// TIA Portal V19 export
FUNCTION_BLOCK "Generic_FB"   // FB108, LAD
TITLE = GENERIC STUFF OF AREA 01 CONTROL CABINET
// stored: Access Published, MemoryReserve 100, SetENOAutomatically false
   VAR_INPUT
      AreaInterface1 : "AreaInterface";
      AreaInterface2 : "AreaInterface";
      AreaInterface3 : "AreaInterface";
      AreaInterface4 : "AreaInterface";
   END_VAR
   VAR_OUTPUT
      MachineInterface1 : "MachineInterface";
      MachineInterface2 : "MachineInterface";
      MachineInterface3 : "MachineInterface";
      MachineInterface4 : "MachineInterface";
   END_VAR
   VAR
      Ctrl : Struct
         RstAlarms : Bool;
      END_STRUCT;
      Sts : Struct
         Standstill : Bool := TRUE;
         AlarmsPresence_GEN : Bool := FALSE;
         AlarmsPresence_A01_2 : Bool;
         AlarmsPresence_A03_4 : Bool;
         WarningsPresence : Bool := FALSE;
      END_STRUCT;
      Alarm : Struct
         CC1_PorteAperte : Bool;
         CC1_ThermalTrip_24Vdc_PLC_SINAMICS : Bool;
         CC1_ThermalTrip_24Vdc_Valves : Bool;
         CC1_ProtezioneElettronicaSitop : Bool;
         CC1_LowAirPressure : Bool;
         Area01_Aspo_LowAirPressure : Bool;
         Area02_03_Accopiamento_LowAirPressure : Bool;
         Area03_Pareggiamneto_LowAirPressure : Bool;
         Area04_Navetta_LowAirPressure : Bool;
         INFEED_640A1 : "InfeedAlr";
         CU_580A1 : "SinamicsCU_Alarms";
         CU_585A1 : "SinamicsCU_Alarms";
         CU_590A1 : "SinamicsCU_Alarms";
         CU_595A1 : "SinamicsCU_Alarms";
         CU_600A1 : "SinamicsCU_Alarms";
         CU_605A1 : "SinamicsCU_Alarms";
         CU_610A1 : "SinamicsCU_Alarms";
         CU_615A1 : "SinamicsCU_Alarms";
         PNDiag_ET200S_460A1 : "PnDiag_Alr";
         PNDiag_ET200S_490A1 : "PnDiag_Alr";
         PNDiag_ET200S_510A1 : "PnDiag_Alr";
         PNDiag_ET200S_530A1 : "PnDiag_Alr";
         PNDiag_ET200S_550A1 : "PnDiag_Alr";
         PNDiag_CU_580A1 : "PnDiag_Alr";
         PNDiag_CU_585A1 : "PnDiag_Alr";
         PNDiag_CU_590A1 : "PnDiag_Alr";
         PNDiag_CU_595A1 : "PnDiag_Alr";
         PNDiag_CU_600A1 : "PnDiag_Alr";
         PNDiag_CU_605A1 : "PnDiag_Alr";
         PNDiag_CU_610A1 : "PnDiag_Alr";
         PNDiag_CU_615A1 : "PnDiag_Alr";
         PnDiag_ENC_694P1 { S7_SetPoint := 'True'} : "PnDiag_Alr";
         PnDiag_ENC_894P1 { S7_SetPoint := 'True'} : "PnDiag_Alr";
         PnDiag_ENC_984P1 { S7_SetPoint := 'True'} : "PnDiag_Alr";
         PnDiag_ENC_994P1 { S7_SetPoint := 'True'} : "PnDiag_Alr";
         PnDiag_ENC_1004P1 { S7_SetPoint := 'True'} : "PnDiag_Alr";
         PnDiag_ENC_1008P1 { S7_SetPoint := 'True'} : "PnDiag_Alr";
         PnDiag_ENC_1034P1 { S7_SetPoint := 'True'} : "PnDiag_Alr";
         PnDiag_ENC_1044P1 { S7_SetPoint := 'True'} : "PnDiag_Alr";
         PnDiag_ENC_1074P1 { S7_SetPoint := 'True'} : "PnDiag_Alr";
         PnDiag_ENC_1088P1 { S7_SetPoint := 'True'} : "PnDiag_Alr";
         PnDiag_ENC_1093P1 { S7_SetPoint := 'True'} : "PnDiag_Alr";
         PnDiag_ENC_1124P1 { S7_SetPoint := 'True'} : "PnDiag_Alr";
         PnDiag_ENC_1138P1 { S7_SetPoint := 'True'} : "PnDiag_Alr";
         PnDiag_ENC_1143P1 { S7_SetPoint := 'True'} : "PnDiag_Alr";
         PnDiag_ENC_1844P1 { S7_SetPoint := 'True'} : "PnDiag_Alr";
         PnDiag_ENC_1853P1 { S7_SetPoint := 'True'} : "PnDiag_Alr";
         PnDiag_ENC_1858P1 { S7_SetPoint := 'True'} : "PnDiag_Alr";
         PnDiag_ENC_1863P1 { S7_SetPoint := 'True'} : "PnDiag_Alr";
         PnDiag_ENC_1868P1 { S7_SetPoint := 'True'} : "PnDiag_Alr";
         PnDiag_ENC_1903P1 { S7_SetPoint := 'True'} : "PnDiag_Alr";
         PnDiag_ENC_1908P1 { S7_SetPoint := 'True'} : "PnDiag_Alr";
         PnDiag_ENC_1913P1 { S7_SetPoint := 'True'} : "PnDiag_Alr";
         PnDiag_ENC_1918P1 { S7_SetPoint := 'True'} : "PnDiag_Alr";
         PnDiag_ENC_2264P1 { S7_SetPoint := 'True'} : "PnDiag_Alr";
         PnDiag_ENC_2284P1 { S7_SetPoint := 'True'} : "PnDiag_Alr";
         PnDiag_ENC_2374P1 { S7_SetPoint := 'True'} : "PnDiag_Alr";
         PnDiag_ENC_2394P1 { S7_SetPoint := 'True'} : "PnDiag_Alr";
         PnDiag_ENC_2404P1 { S7_SetPoint := 'True'} : "PnDiag_Alr";
         PnDiag_ENC_2434P1 { S7_SetPoint := 'True'} : "PnDiag_Alr";
         PnDiag_ENC_2464P1 { S7_SetPoint := 'True'} : "PnDiag_Alr";
         PnDiag_ENC_2534P1 { S7_SetPoint := 'True'} : "PnDiag_Alr";
         PnDiag_PAC_100A1 { S7_SetPoint := 'True'} : "PnDiag_Alr";
      END_STRUCT;
      Warning : Struct
         NoAutReady : Bool;
         CC1_ThermalTrip220V_ServiceSockets : Bool;
         CC1_ThermalTrip_Cooling1 : Bool;
         CC1_ThermalTrip_Cooling2 : Bool;
         JB001_ThermalTrip_Cooling : Bool;
         CC1_MaxTemperature : Bool;
         JB001_MaxTemperature : Bool;
         CC1_GuastoCondizionatore_1 : Bool;
         CC1_GuastoCondizionatore_2 : Bool;
         SitopUp_BatteriaScarica : Bool;
         SitopUp_BatteriaNonCarica : Bool;
         SitopUp_AllarmeBatteria : Bool;
         ScalanceXC116_1_NotOk : Bool;
         ScalanceXC116_2_NotOk : Bool;
         ScalanceXC216_NotOk : Bool;
         ScalanceSC632_NotOk : Bool;
         INFEED_640A1 : "InfeedWng";
         CU_580A1 : "SinamicsCU_Warnings";
         CU_585A1 : "SinamicsCU_Warnings";
         CU_590A1 : "SinamicsCU_Warnings";
         CU_595A1 : "SinamicsCU_Warnings";
         CU_600A1 : "SinamicsCU_Warnings";
         CU_605A1 : "SinamicsCU_Warnings";
         CU_610A1 : "SinamicsCU_Warnings";
         CU_615A1 : "SinamicsCU_Warnings";
      END_STRUCT;
      Diag : Struct
         CC1_INFEED_460A1 : "TO_Diagnostic";
         CU_580A1 { S7_SetPoint := 'True'} : "TO_Diagnostic";
         CU_585A1 { S7_SetPoint := 'True'} : "TO_Diagnostic";
         CU_590A1 { S7_SetPoint := 'True'} : "TO_Diagnostic";
         CU_595A1 { S7_SetPoint := 'True'} : "TO_Diagnostic";
         CU_600A1 { S7_SetPoint := 'True'} : "TO_Diagnostic";
         CU_605A1 { S7_SetPoint := 'True'} : "TO_Diagnostic";
         CU_610A1 { S7_SetPoint := 'True'} : "TO_Diagnostic";
         CU_615A1 { S7_SetPoint := 'True'} : "TO_Diagnostic";
      END_STRUCT;
      INFEED_640A1 : "Infeed";
      CU_580A1 : "SinamicsCU_Modulblock";
      CU_585A1 : "SinamicsCU_Modulblock";
      CU_590A1 : "SinamicsCU_Modulblock";
      CU_595A1 : "SinamicsCU_Modulblock";
      CU_600A1 : "SinamicsCU_Modulblock";
      CU_605A1 : "SinamicsCU_Modulblock";
      CU_610A1 : "SinamicsCU_Modulblock";
      CU_615A1 : "SinamicsCU_Modulblock";
      PnDiag_ET200S_460A1 : "PnDiag";
      PnDiag_ET200S_490A1 : "PnDiag";
      PnDiag_ET200S_510A1 : "PnDiag";
      PnDiag_ET200S_530A1 : "PnDiag";
      PnDiag_ET200S_550A1 : "PnDiag";
      PnDiag_CU_580A1 : "PnDiag";
      PnDiag_CU_585A1 : "PnDiag";
      PnDiag_CU_590A1 : "PnDiag";
      PnDiag_CU_595A1 : "PnDiag";
      PnDiag_CU_600A1 : "PnDiag";
      PnDiag_CU_605A1 : "PnDiag";
      PnDiag_CU_610A1 : "PnDiag";
      PnDiag_CU_615A1 : "PnDiag";
      PnDiag_ENC_694P1 { S7_SetPoint := 'True'} : "PnDiag";
      PnDiag_ENC_894P1 { S7_SetPoint := 'True'} : "PnDiag";
      PnDiag_ENC_984P1 { S7_SetPoint := 'True'} : "PnDiag";
      PnDiag_ENC_994P1 { S7_SetPoint := 'True'} : "PnDiag";
      PnDiag_ENC_1004P1 { S7_SetPoint := 'True'} : "PnDiag";
      PnDiag_ENC_1008P1 { S7_SetPoint := 'True'} : "PnDiag";
      PnDiag_ENC_1034P1 { S7_SetPoint := 'True'} : "PnDiag";
      PnDiag_ENC_1044P1 { S7_SetPoint := 'True'} : "PnDiag";
      PnDiag_ENC_1074P1 { S7_SetPoint := 'True'} : "PnDiag";
      PnDiag_ENC_1088P1 { S7_SetPoint := 'True'} : "PnDiag";
      PnDiag_ENC_1093P1 { S7_SetPoint := 'True'} : "PnDiag";
      PnDiag_ENC_1124P1 { S7_SetPoint := 'True'} : "PnDiag";
      PnDiag_ENC_1138P1 { S7_SetPoint := 'True'} : "PnDiag";
      PnDiag_ENC_1143P1 { S7_SetPoint := 'True'} : "PnDiag";
      PnDiag_ENC_1844P1 { S7_SetPoint := 'True'} : "PnDiag";
      PnDiag_ENC_1853P1 { S7_SetPoint := 'True'} : "PnDiag";
      PnDiag_ENC_1858P1 { S7_SetPoint := 'True'} : "PnDiag";
      PnDiag_ENC_1863P1 { S7_SetPoint := 'True'} : "PnDiag";
      PnDiag_ENC_1868P1 { S7_SetPoint := 'True'} : "PnDiag";
      PnDiag_ENC_1903P1 { S7_SetPoint := 'True'} : "PnDiag";
      PnDiag_ENC_1908P1 { S7_SetPoint := 'True'} : "PnDiag";
      PnDiag_ENC_1913P1 { S7_SetPoint := 'True'} : "PnDiag";
      PnDiag_ENC_1918P1 { S7_SetPoint := 'True'} : "PnDiag";
      PnDiag_ENC_2264P1 { S7_SetPoint := 'True'} : "PnDiag";
      PnDiag_ENC_2284P1 { S7_SetPoint := 'True'} : "PnDiag";
      PnDiag_ENC_2374P1 { S7_SetPoint := 'True'} : "PnDiag";
      PnDiag_ENC_2394P1 { S7_SetPoint := 'True'} : "PnDiag";
      PnDiag_ENC_2404P1 { S7_SetPoint := 'True'} : "PnDiag";
      PnDiag_ENC_2434P1 { S7_SetPoint := 'True'} : "PnDiag";
      PnDiag_ENC_2464P1 { S7_SetPoint := 'True'} : "PnDiag";
      PnDiag_ENC_2534P1 { S7_SetPoint := 'True'} : "PnDiag";
      PnDiag_PAC_100A1 { S7_SetPoint := 'True'} : "PnDiag";
      TON_CheckHighTemperatureCC1 : IEC_TIMER;
      TON_CheckHighTemperatureJB001 : IEC_TIMER;
      TOF_TurnOffConditionerCC1 : IEC_TIMER;
      TOF_TurnOffConditionerJB001 : IEC_TIMER;
      TON_Area02_03_Accoppiamento_Pressione_Aria_OK { S7_SetPoint := 'True'} : IEC_TIMER;
      TON_Area03_Pareggiamneto_Pressione_Aria_OK { S7_SetPoint := 'True'} : IEC_TIMER;
      TON_Area04_Navetta_Pressione_Aria_OK { S7_SetPoint := 'True'} : IEC_TIMER;
   END_VAR
   VAR CONSTANT
      MSG_A1073_POWER_ON_REQ_BACKUP_COPY : UInt := 1073;
      MSG_A13030_TRIAL_LICENSE_ACTIVATE : UInt := 13030;
   END_VAR
BEGIN

REGION Network 1: Reset alarms
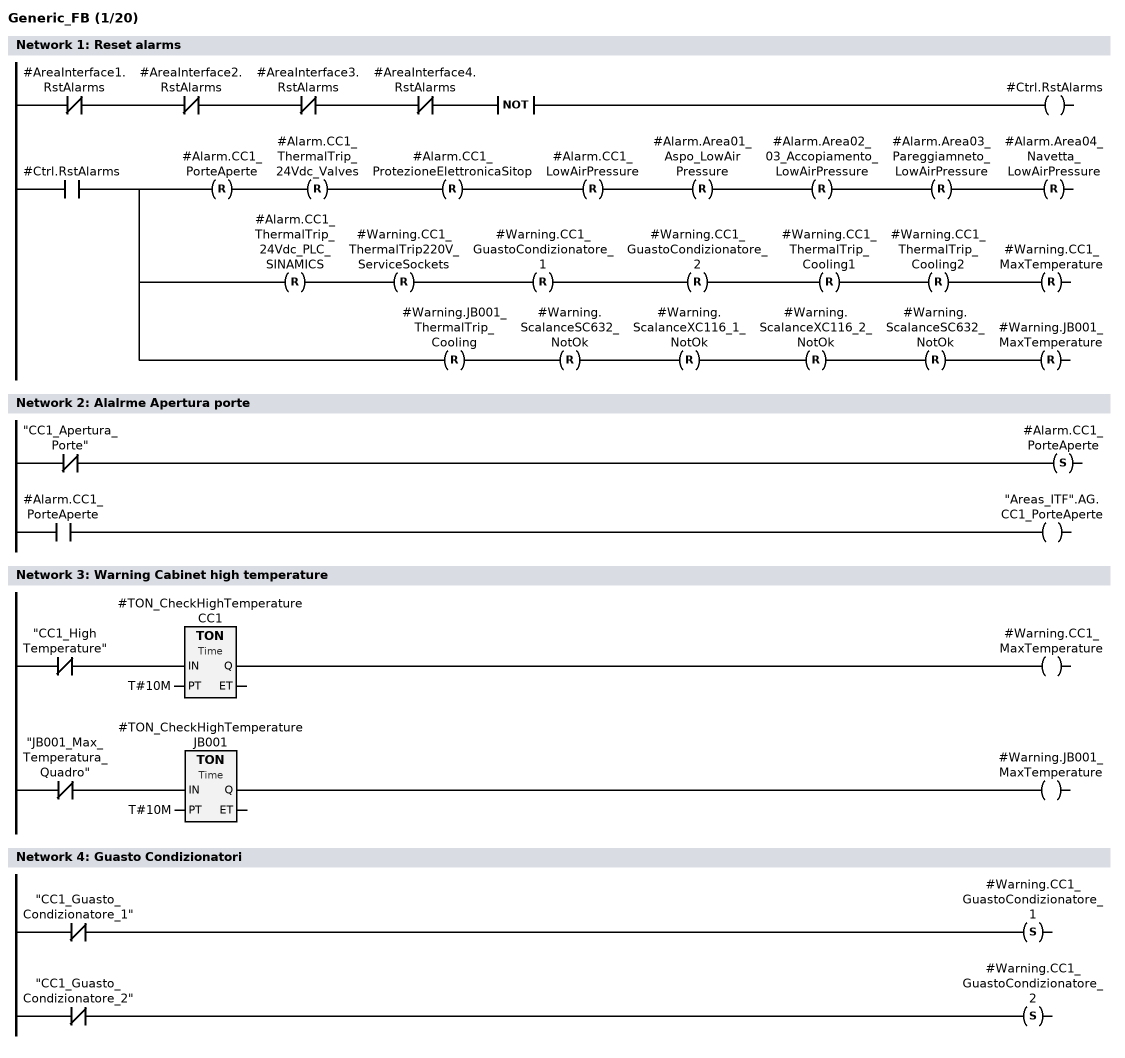
   RUNG wire#powerrail
      I_Contact( #AreaInterface1.RstAlarms )
      I_Contact( #AreaInterface2.RstAlarms )
      I_Contact( #AreaInterface3.RstAlarms )
      I_Contact( #AreaInterface4.RstAlarms )
      Not()
      Coil( #Ctrl.RstAlarms )
   END_RUNG
   RUNG wire#powerrail
      Contact( #Ctrl.RstAlarms )
      wire#w1
      R_Coil( #Alarm.CC1_PorteAperte )
      R_Coil( #Alarm.CC1_ThermalTrip_24Vdc_Valves )
      R_Coil( #Alarm.CC1_ProtezioneElettronicaSitop )
      R_Coil( #Alarm.CC1_LowAirPressure )
      R_Coil( #Alarm.Area01_Aspo_LowAirPressure )
      R_Coil( #Alarm.Area02_03_Accopiamento_LowAirPressure )
      R_Coil( #Alarm.Area03_Pareggiamneto_LowAirPressure )
      R_Coil( #Alarm.Area04_Navetta_LowAirPressure )
   END_RUNG
   RUNG wire#w1
      R_Coil( #Alarm.CC1_ThermalTrip_24Vdc_PLC_SINAMICS )
      R_Coil( #Warning.CC1_ThermalTrip220V_ServiceSockets )
      R_Coil( #Warning.CC1_GuastoCondizionatore_1 )
      R_Coil( #Warning.CC1_GuastoCondizionatore_2 )
      R_Coil( #Warning.CC1_ThermalTrip_Cooling1 )
      R_Coil( #Warning.CC1_ThermalTrip_Cooling2 )
      R_Coil( #Warning.CC1_MaxTemperature )
   END_RUNG
   RUNG wire#w1
      R_Coil( #Warning.JB001_ThermalTrip_Cooling )
      R_Coil( #Warning.ScalanceSC632_NotOk )
      R_Coil( #Warning.ScalanceXC116_1_NotOk )
      R_Coil( #Warning.ScalanceXC116_2_NotOk )
      R_Coil( #Warning.ScalanceSC632_NotOk )
      R_Coil( #Warning.JB001_MaxTemperature )
   END_RUNG
   // the same network as SCL:
   #Ctrl.RstAlarms := NOT (NOT #AreaInterface1.RstAlarms AND NOT #AreaInterface2.RstAlarms AND NOT #AreaInterface3.RstAlarms AND NOT #AreaInterface4.RstAlarms);
   IF #Ctrl.RstAlarms THEN
       #Alarm.CC1_PorteAperte := FALSE;
       #Alarm.CC1_ThermalTrip_24Vdc_Valves := FALSE;
       #Alarm.CC1_ProtezioneElettronicaSitop := FALSE;
       #Alarm.CC1_LowAirPressure := FALSE;
       #Alarm.Area01_Aspo_LowAirPressure := FALSE;
       #Alarm.Area02_03_Accopiamento_LowAirPressure := FALSE;
       #Alarm.Area03_Pareggiamneto_LowAirPressure := FALSE;
       #Alarm.Area04_Navetta_LowAirPressure := FALSE;
       #Alarm.CC1_ThermalTrip_24Vdc_PLC_SINAMICS := FALSE;
       #Warning.CC1_ThermalTrip220V_ServiceSockets := FALSE;
       #Warning.CC1_GuastoCondizionatore_1 := FALSE;
       #Warning.CC1_GuastoCondizionatore_2 := FALSE;
       #Warning.CC1_ThermalTrip_Cooling1 := FALSE;
       #Warning.CC1_ThermalTrip_Cooling2 := FALSE;
       #Warning.CC1_MaxTemperature := FALSE;
       #Warning.JB001_ThermalTrip_Cooling := FALSE;
       #Warning.ScalanceSC632_NotOk := FALSE;
       #Warning.ScalanceXC116_1_NotOk := FALSE;
       #Warning.ScalanceXC116_2_NotOk := FALSE;
       #Warning.ScalanceSC632_NotOk := FALSE;
       #Warning.JB001_MaxTemperature := FALSE;
   END_IF;
END_REGION

REGION Network 2: Alalrme Apertura porte
   RUNG wire#powerrail
      I_Contact( "CC1_Apertura_Porte" )
      S_Coil( #Alarm.CC1_PorteAperte )
   END_RUNG
   RUNG wire#powerrail
      Contact( #Alarm.CC1_PorteAperte )
      Coil( "Areas_ITF".AG.CC1_PorteAperte )
   END_RUNG
   // the same network as SCL:
   IF NOT "CC1_Apertura_Porte" THEN #Alarm.CC1_PorteAperte := TRUE; END_IF;
   "Areas_ITF".AG.CC1_PorteAperte := #Alarm.CC1_PorteAperte;
END_REGION

REGION Network 3: Warning Cabinet high temperature
   RUNG wire#powerrail
      I_Contact( "CC1_HighTemperature" )
      { S7_Templates := "time_type := Time" } #TON_CheckHighTemperatureCC1.TON(pt := T#10M, et =>)
      Coil( #Warning.CC1_MaxTemperature )
   END_RUNG
   RUNG wire#powerrail
      I_Contact( "JB001_Max_Temperatura_Quadro" )
      { S7_Templates := "time_type := Time" } #TON_CheckHighTemperatureJB001.TON(pt := T#10M, et =>)
      Coil( #Warning.JB001_MaxTemperature )
   END_RUNG
   // the same network as SCL:
   #TON_CheckHighTemperatureCC1.TON(IN := NOT "CC1_HighTemperature", PT := T#10M);
   #Warning.CC1_MaxTemperature := #TON_CheckHighTemperatureCC1.Q;
   #TON_CheckHighTemperatureJB001.TON(IN := NOT "JB001_Max_Temperatura_Quadro", PT := T#10M);
   #Warning.JB001_MaxTemperature := #TON_CheckHighTemperatureJB001.Q;
END_REGION

REGION Network 4: Guasto Condizionatori
   RUNG wire#powerrail
      I_Contact( "CC1_Guasto_Condizionatore_1" )
      S_Coil( #Warning.CC1_GuastoCondizionatore_1 )
   END_RUNG
   RUNG wire#powerrail
      I_Contact( "CC1_Guasto_Condizionatore_2" )
      S_Coil( #Warning.CC1_GuastoCondizionatore_2 )
   END_RUNG
   // the same network as SCL:
   IF NOT "CC1_Guasto_Condizionatore_1" THEN #Warning.CC1_GuastoCondizionatore_1 := TRUE; END_IF;
   IF NOT "CC1_Guasto_Condizionatore_2" THEN #Warning.CC1_GuastoCondizionatore_2 := TRUE; END_IF;
END_REGION

REGION Network 5: Comando Condizionatori
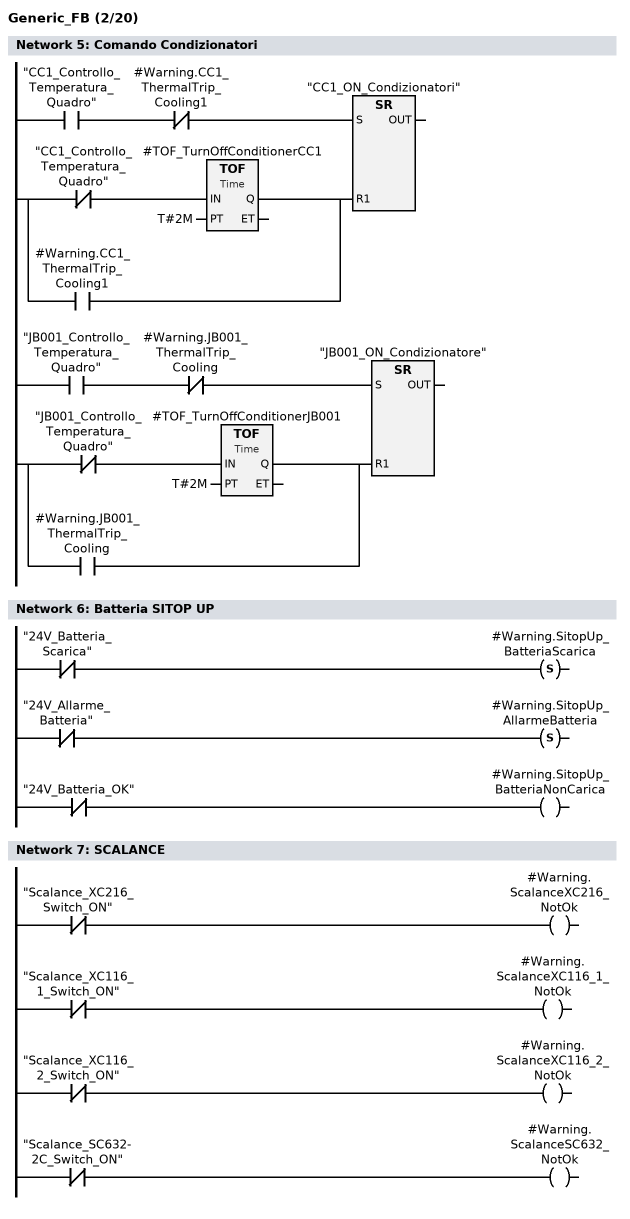
   RUNG wire#powerrail
      Contact( "CC1_Controllo_Temperatura_Quadro" )
      I_Contact( #Warning.CC1_ThermalTrip_Cooling1 )
      S_SR(operand := "CC1_ON_Condizionatori", r1 := wire#w1)
   END_RUNG
   RUNG wire#powerrail
      I_Contact( "CC1_Controllo_Temperatura_Quadro" )
      { S7_Templates := "time_type := Time" } #TOF_TurnOffConditionerCC1.TOF(pt := T#2M, et =>)
   END_RUNG wire#w1
   RUNG wire#powerrail
      Contact( #Warning.CC1_ThermalTrip_Cooling1 )
   END_RUNG wire#w1
   RUNG wire#powerrail
      Contact( "JB001_Controllo_Temperatura_Quadro" )
      I_Contact( #Warning.JB001_ThermalTrip_Cooling )
      S_SR(operand := "JB001_ON_Condizionatore", r1 := wire#w2)
   END_RUNG
   RUNG wire#powerrail
      I_Contact( "JB001_Controllo_Temperatura_Quadro" )
      { S7_Templates := "time_type := Time" } #TOF_TurnOffConditionerJB001.TOF(pt := T#2M, et =>)
   END_RUNG wire#w2
   RUNG wire#powerrail
      Contact( #Warning.JB001_ThermalTrip_Cooling )
   END_RUNG wire#w2
   // the same network as SCL:
   #TOF_TurnOffConditionerCC1.TOF(IN := NOT "CC1_Controllo_Temperatura_Quadro", PT := T#2M);
   IF "CC1_Controllo_Temperatura_Quadro" AND NOT #Warning.CC1_ThermalTrip_Cooling1 THEN
       "CC1_ON_Condizionatori" := TRUE;   // SR flip-flop
   END_IF;
   IF #TOF_TurnOffConditionerCC1.Q OR #Warning.CC1_ThermalTrip_Cooling1 THEN
       "CC1_ON_Condizionatori" := FALSE;
   END_IF;
   #TOF_TurnOffConditionerJB001.TOF(IN := NOT "JB001_Controllo_Temperatura_Quadro", PT := T#2M);
   IF "JB001_Controllo_Temperatura_Quadro" AND NOT #Warning.JB001_ThermalTrip_Cooling THEN
       "JB001_ON_Condizionatore" := TRUE;   // SR flip-flop
   END_IF;
   IF #TOF_TurnOffConditionerJB001.Q OR #Warning.JB001_ThermalTrip_Cooling THEN
       "JB001_ON_Condizionatore" := FALSE;
   END_IF;
END_REGION

REGION Network 6: Batteria SITOP UP
   RUNG wire#powerrail
      I_Contact( "24V_Batteria_Scarica" )
      S_Coil( #Warning.SitopUp_BatteriaScarica )
   END_RUNG
   RUNG wire#powerrail
      I_Contact( "24V_Allarme_Batteria" )
      S_Coil( #Warning.SitopUp_AllarmeBatteria )
   END_RUNG
   RUNG wire#powerrail
      I_Contact( "24V_Batteria_OK" )
      Coil( #Warning.SitopUp_BatteriaNonCarica )
   END_RUNG
   // the same network as SCL:
   IF NOT "24V_Batteria_Scarica" THEN #Warning.SitopUp_BatteriaScarica := TRUE; END_IF;
   IF NOT "24V_Allarme_Batteria" THEN #Warning.SitopUp_AllarmeBatteria := TRUE; END_IF;
   #Warning.SitopUp_BatteriaNonCarica := NOT "24V_Batteria_OK";
END_REGION

REGION Network 7: SCALANCE
   RUNG wire#powerrail
      I_Contact( "Scalance_XC216_Switch_ON" )
      Coil( #Warning.ScalanceXC216_NotOk )
   END_RUNG
   RUNG wire#powerrail
      I_Contact( "Scalance_XC116_1_Switch_ON" )
      Coil( #Warning.ScalanceXC116_1_NotOk )
   END_RUNG
   RUNG wire#powerrail
      I_Contact( "Scalance_XC116_2_Switch_ON" )
      Coil( #Warning.ScalanceXC116_2_NotOk )
   END_RUNG
   RUNG wire#powerrail
      I_Contact( "Scalance_SC632-2C_Switch_ON" )
      Coil( #Warning.ScalanceSC632_NotOk )
   END_RUNG
   // the same network as SCL:
   #Warning.ScalanceXC216_NotOk := NOT "Scalance_XC216_Switch_ON";
   #Warning.ScalanceXC116_1_NotOk := NOT "Scalance_XC116_1_Switch_ON";
   #Warning.ScalanceXC116_2_NotOk := NOT "Scalance_XC116_2_Switch_ON";
   #Warning.ScalanceSC632_NotOk := NOT "Scalance_SC632-2C_Switch_ON";
END_REGION

REGION Network 8: Alarm Thermal trips
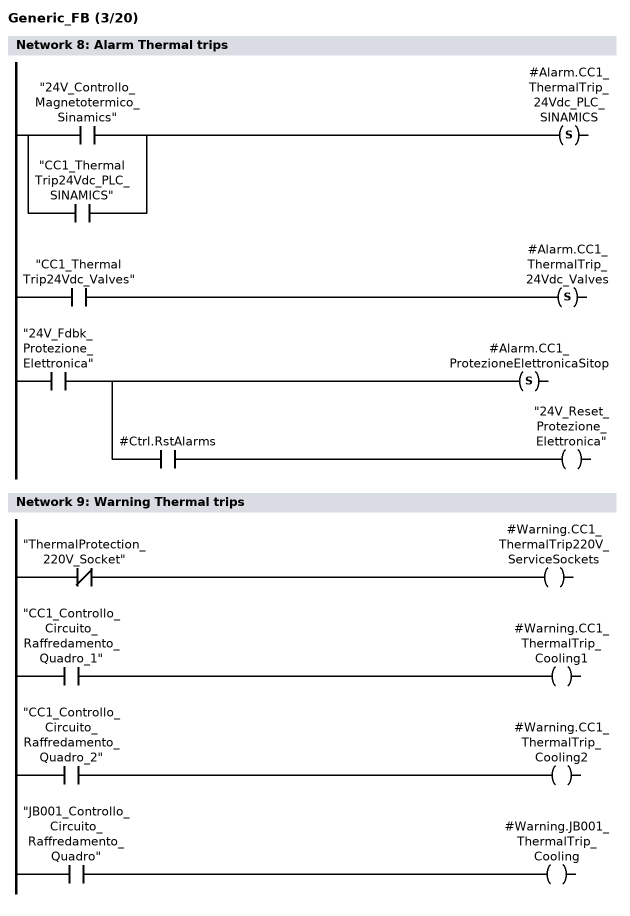
   RUNG wire#powerrail
      Contact( "24V_Controllo_Magnetotermico_Sinamics" )
      wire#w1
      S_Coil( #Alarm.CC1_ThermalTrip_24Vdc_PLC_SINAMICS )
   END_RUNG
   RUNG wire#powerrail
      Contact( "CC1_ThermalTrip24Vdc_PLC_SINAMICS" )
   END_RUNG wire#w1
   RUNG wire#powerrail
      Contact( "CC1_ThermalTrip24Vdc_Valves" )
      S_Coil( #Alarm.CC1_ThermalTrip_24Vdc_Valves )
   END_RUNG
   RUNG wire#powerrail
      Contact( "24V_Fdbk_Protezione_Elettronica" )
      wire#w2
      S_Coil( #Alarm.CC1_ProtezioneElettronicaSitop )
   END_RUNG
   RUNG wire#w2
      Contact( #Ctrl.RstAlarms )
      Coil( "24V_Reset_Protezione_Elettronica" )
   END_RUNG
   // the same network as SCL:
   IF "24V_Controllo_Magnetotermico_Sinamics" OR "CC1_ThermalTrip24Vdc_PLC_SINAMICS" THEN
       #Alarm.CC1_ThermalTrip_24Vdc_PLC_SINAMICS := TRUE;
   END_IF;
   IF "CC1_ThermalTrip24Vdc_Valves" THEN #Alarm.CC1_ThermalTrip_24Vdc_Valves := TRUE; END_IF;
   IF "24V_Fdbk_Protezione_Elettronica" THEN #Alarm.CC1_ProtezioneElettronicaSitop := TRUE; END_IF;
   "24V_Reset_Protezione_Elettronica" := "24V_Fdbk_Protezione_Elettronica" AND #Ctrl.RstAlarms;
END_REGION

REGION Network 9: Warning Thermal trips
   RUNG wire#powerrail
      I_Contact( "ThermalProtection_220V_Socket" )
      Coil( #Warning.CC1_ThermalTrip220V_ServiceSockets )
   END_RUNG
   RUNG wire#powerrail
      Contact( "CC1_Controllo_Circuito_Raffredamento_Quadro_1" )
      Coil( #Warning.CC1_ThermalTrip_Cooling1 )
   END_RUNG
   RUNG wire#powerrail
      Contact( "CC1_Controllo_Circuito_Raffredamento_Quadro_2" )
      Coil( #Warning.CC1_ThermalTrip_Cooling2 )
   END_RUNG
   RUNG wire#powerrail
      Contact( "JB001_Controllo_Circuito_Raffredamento_Quadro" )
      Coil( #Warning.JB001_ThermalTrip_Cooling )
   END_RUNG
   // the same network as SCL:
   #Warning.CC1_ThermalTrip220V_ServiceSockets := NOT "ThermalProtection_220V_Socket";
   #Warning.CC1_ThermalTrip_Cooling1 := "CC1_Controllo_Circuito_Raffredamento_Quadro_1";
   #Warning.CC1_ThermalTrip_Cooling2 := "CC1_Controllo_Circuito_Raffredamento_Quadro_2";
   #Warning.JB001_ThermalTrip_Cooling := "JB001_Controllo_Circuito_Raffredamento_Quadro";
END_REGION

REGION Network 10: Alarm Low air pressure
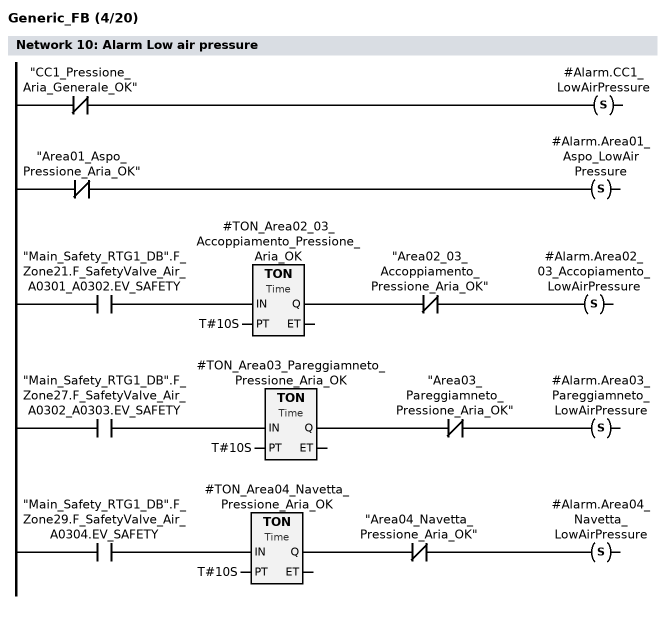
   RUNG wire#powerrail
      I_Contact( "CC1_Pressione_Aria_Generale_OK" )
      S_Coil( #Alarm.CC1_LowAirPressure )
   END_RUNG
   RUNG wire#powerrail
      I_Contact( "Area01_Aspo_Pressione_Aria_OK" )
      S_Coil( #Alarm.Area01_Aspo_LowAirPressure )
   END_RUNG
   RUNG wire#powerrail
      Contact( "Main_Safety_RTG1_DB".F_Zone21.F_SafetyValve_Air_A0301_A0302.EV_SAFETY )
      { S7_Templates := "time_type := Time" } #TON_Area02_03_Accoppiamento_Pressione_Aria_OK.TON(pt := T#10S, et =>)
      I_Contact( "Area02_03_Accoppiamento_Pressione_Aria_OK" )
      S_Coil( #Alarm.Area02_03_Accopiamento_LowAirPressure )
   END_RUNG
   RUNG wire#powerrail
      Contact( "Main_Safety_RTG1_DB".F_Zone27.F_SafetyValve_Air_A0302_A0303.EV_SAFETY )
      { S7_Templates := "time_type := Time" } #TON_Area03_Pareggiamneto_Pressione_Aria_OK.TON(pt := T#10S, et =>)
      I_Contact( "Area03_Pareggiamneto_Pressione_Aria_OK" )
      S_Coil( #Alarm.Area03_Pareggiamneto_LowAirPressure )
   END_RUNG
   RUNG wire#powerrail
      Contact( "Main_Safety_RTG1_DB".F_Zone29.F_SafetyValve_Air_A0304.EV_SAFETY )
      { S7_Templates := "time_type := Time" } #TON_Area04_Navetta_Pressione_Aria_OK.TON(pt := T#10S, et =>)
      I_Contact( "Area04_Navetta_Pressione_Aria_OK" )
      S_Coil( #Alarm.Area04_Navetta_LowAirPressure )
   END_RUNG
   // the same network as SCL:
   IF NOT "CC1_Pressione_Aria_Generale_OK" THEN #Alarm.CC1_LowAirPressure := TRUE; END_IF;
   IF NOT "Area01_Aspo_Pressione_Aria_OK" THEN #Alarm.Area01_Aspo_LowAirPressure := TRUE; END_IF;
   #TON_Area02_03_Accoppiamento_Pressione_Aria_OK.TON(IN := "Main_Safety_RTG1_DB".F_Zone21.F_SafetyValve_Air_A0301_A0302.EV_SAFETY,
                           PT := T#10S);
   IF #TON_Area02_03_Accoppiamento_Pressione_Aria_OK.Q AND NOT "Area02_03_Accoppiamento_Pressione_Aria_OK" THEN
       #Alarm.Area02_03_Accopiamento_LowAirPressure := TRUE;
   END_IF;
   #TON_Area03_Pareggiamneto_Pressione_Aria_OK.TON(IN := "Main_Safety_RTG1_DB".F_Zone27.F_SafetyValve_Air_A0302_A0303.EV_SAFETY,
                           PT := T#10S);
   IF #TON_Area03_Pareggiamneto_Pressione_Aria_OK.Q AND NOT "Area03_Pareggiamneto_Pressione_Aria_OK" THEN
       #Alarm.Area03_Pareggiamneto_LowAirPressure := TRUE;
   END_IF;
   #TON_Area04_Navetta_Pressione_Aria_OK.TON(IN := "Main_Safety_RTG1_DB".F_Zone29.F_SafetyValve_Air_A0304.EV_SAFETY,
                           PT := T#10S);
   IF #TON_Area04_Navetta_Pressione_Aria_OK.Q AND NOT "Area04_Navetta_Pressione_Aria_OK" THEN
       #Alarm.Area04_Navetta_LowAirPressure := TRUE;
   END_IF;
END_REGION

REGION Network 12: <<< DRIVES >>>
END_REGION

REGION Network 13: Infeed
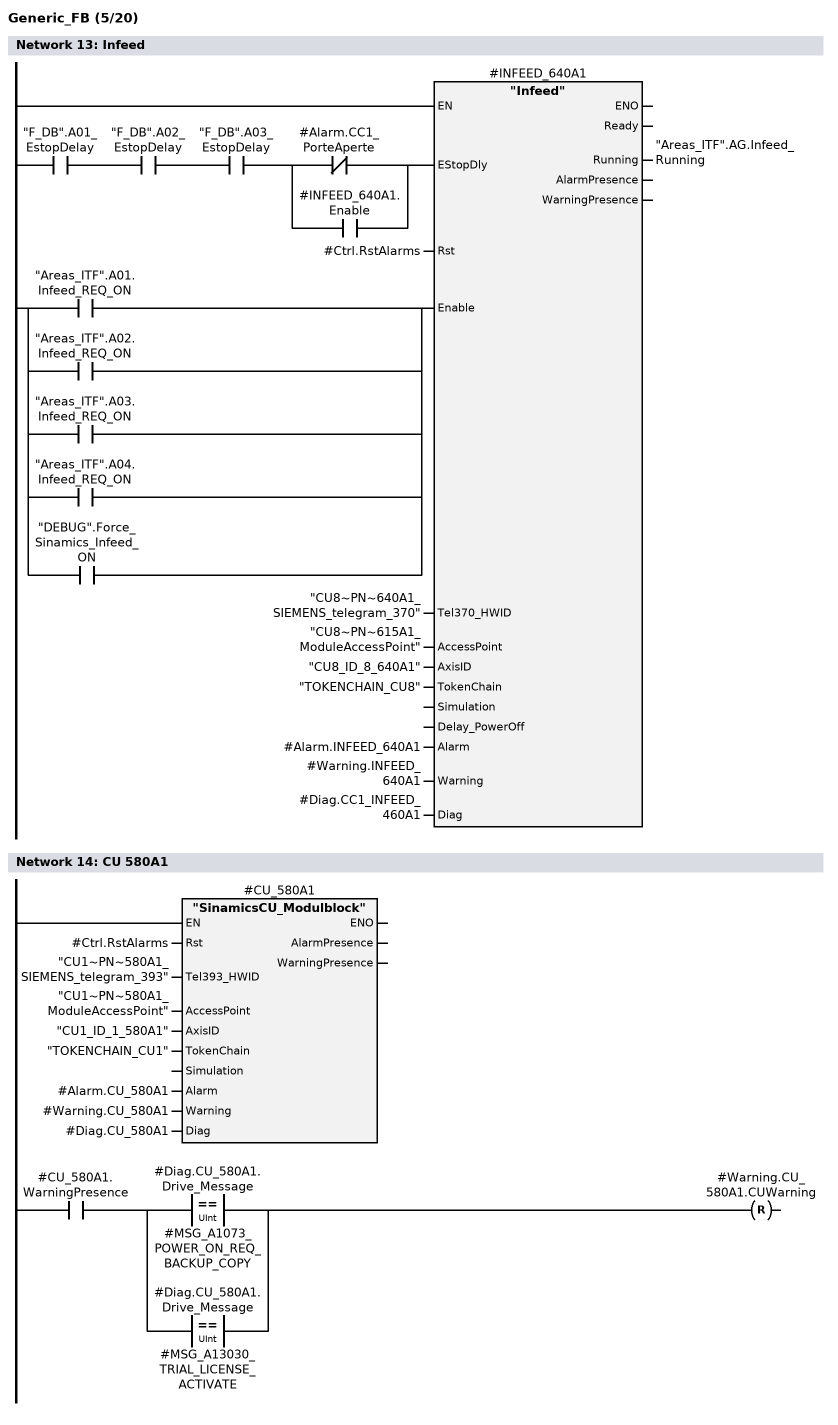
   RUNG wire#powerrail
      #INFEED_640A1(EStopDly := wire#w2, Enable := wire#w3, Rst := #Ctrl.RstAlarms, Tel370_HWID := "CU8~PN~640A1_SIEMENS_telegram_370", AccessPoint := "CU8~PN~615A1_ModuleAccessPoint", AxisID := "CU8_ID_8_640A1", TokenChain := "TOKENCHAIN_CU8", Simulation :=, Delay_PowerOff :=, Alarm := #Alarm.INFEED_640A1, Warning := #Warning.INFEED_640A1, Diag := #Diag.CC1_INFEED_460A1, Ready =>, Running => "Areas_ITF".AG.Infeed_Running, AlarmPresence =>, WarningPresence =>)
   END_RUNG
   RUNG wire#powerrail
      Contact( "F_DB".A01_EstopDelay )
      Contact( "F_DB".A02_EstopDelay )
      Contact( "F_DB".A03_EstopDelay )
      wire#w1
      I_Contact( #Alarm.CC1_PorteAperte )
   END_RUNG wire#w2
   RUNG wire#w1
      Contact( #INFEED_640A1.Enable )
   END_RUNG wire#w2
   RUNG wire#powerrail
      Contact( "Areas_ITF".A01.Infeed_REQ_ON )
   END_RUNG wire#w3
   RUNG wire#powerrail
      Contact( "Areas_ITF".A02.Infeed_REQ_ON )
   END_RUNG wire#w3
   RUNG wire#powerrail
      Contact( "Areas_ITF".A03.Infeed_REQ_ON )
   END_RUNG wire#w3
   RUNG wire#powerrail
      Contact( "Areas_ITF".A04.Infeed_REQ_ON )
   END_RUNG wire#w3
   RUNG wire#powerrail
      Contact( "DEBUG".Force_Sinamics_Infeed_ON )
   END_RUNG wire#w3
   // the same network as SCL:
   #INFEED_640A1(EStopDly := "F_DB".A01_EstopDelay AND "F_DB".A02_EstopDelay AND "F_DB".A03_EstopDelay AND (NOT #Alarm.CC1_PorteAperte OR #INFEED_640A1.Enable),   // "Infeed"
                 Rst := #Ctrl.RstAlarms,
                 Enable := "Areas_ITF".A01.Infeed_REQ_ON OR "Areas_ITF".A02.Infeed_REQ_ON OR "Areas_ITF".A03.Infeed_REQ_ON OR "Areas_ITF".A04.Infeed_REQ_ON OR "DEBUG".Force_Sinamics_Infeed_ON,
                 Tel370_HWID := "CU8~PN~640A1_SIEMENS_telegram_370",
                 AccessPoint := "CU8~PN~615A1_ModuleAccessPoint",
                 AxisID := "CU8_ID_8_640A1",
                 TokenChain := "TOKENCHAIN_CU8",
                 Alarm := #Alarm.INFEED_640A1,
                 Warning := #Warning.INFEED_640A1,
                 Diag := #Diag.CC1_INFEED_460A1,
                 Running => "Areas_ITF".AG.Infeed_Running);
END_REGION

REGION Network 14: CU 580A1
   RUNG wire#powerrail
      #CU_580A1(Rst := #Ctrl.RstAlarms, Tel393_HWID := "CU1~PN~580A1_SIEMENS_telegram_393", AccessPoint := "CU1~PN~580A1_ModuleAccessPoint", AxisID := "CU1_ID_1_580A1", TokenChain := "TOKENCHAIN_CU1", Simulation :=, Alarm := #Alarm.CU_580A1, Warning := #Warning.CU_580A1, Diag := #Diag.CU_580A1, AlarmPresence =>, WarningPresence =>)
   END_RUNG
   RUNG wire#powerrail
      Contact( #CU_580A1.WarningPresence )
      wire#w1
      { S7_Templates := "SrcType := UInt" } EQ_Contact(in1 := #Diag.CU_580A1.Drive_Message, in2 := #MSG_A1073_POWER_ON_REQ_BACKUP_COPY)
      wire#w2
      R_Coil( #Warning.CU_580A1.CUWarning )
   END_RUNG
   RUNG wire#w1
      { S7_Templates := "SrcType := UInt" } EQ_Contact(in1 := #Diag.CU_580A1.Drive_Message, in2 := #MSG_A13030_TRIAL_LICENSE_ACTIVATE)
   END_RUNG wire#w2
   // the same network as SCL:
   #CU_580A1(Rst := #Ctrl.RstAlarms,   // "SinamicsCU_Modulblock"
             Tel393_HWID := "CU1~PN~580A1_SIEMENS_telegram_393",
             AccessPoint := "CU1~PN~580A1_ModuleAccessPoint",
             AxisID := "CU1_ID_1_580A1",
             TokenChain := "TOKENCHAIN_CU1",
             Alarm := #Alarm.CU_580A1,
             Warning := #Warning.CU_580A1,
             Diag := #Diag.CU_580A1);
   IF #CU_580A1.WarningPresence AND ((#Diag.CU_580A1.Drive_Message = #MSG_A1073_POWER_ON_REQ_BACKUP_COPY) OR (#Diag.CU_580A1.Drive_Message = #MSG_A13030_TRIAL_LICENSE_ACTIVATE)) THEN
       #Warning.CU_580A1.CUWarning := FALSE;
   END_IF;
END_REGION

REGION Network 15: CU 585A1
   // Bypass message "POWER ON REQUIRED FOR COPY ON MEMORY CARD"
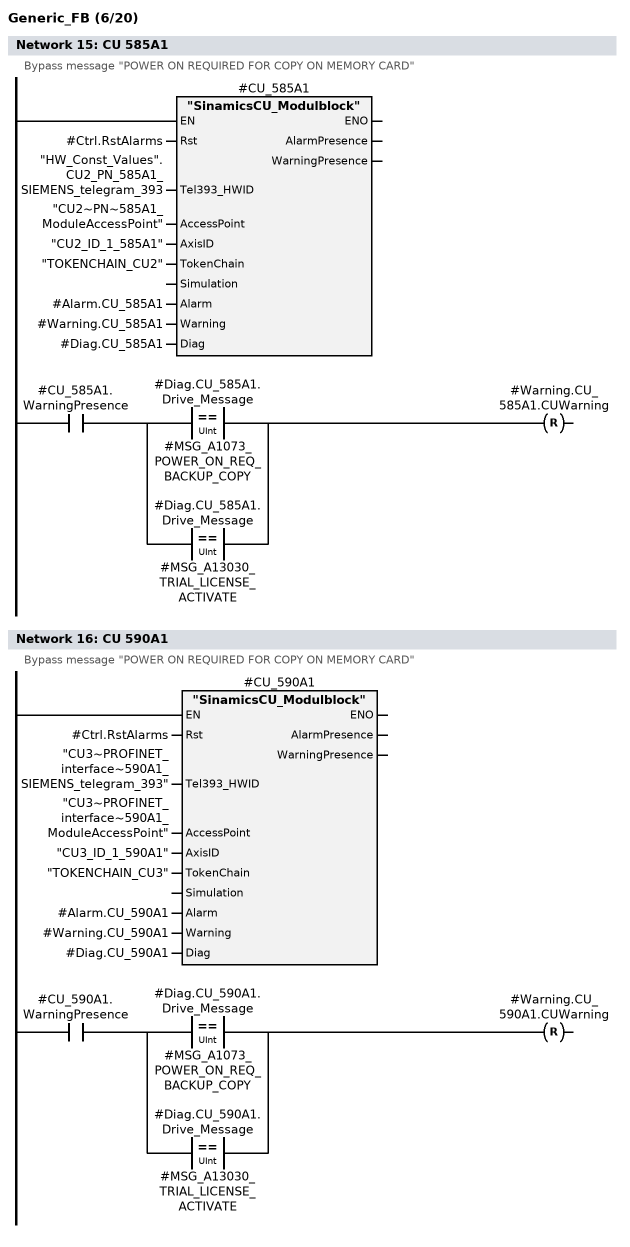
   RUNG wire#powerrail
      #CU_585A1(Rst := #Ctrl.RstAlarms, Tel393_HWID := "HW_Const_Values".CU2_PN_585A1_SIEMENS_telegram_393, AccessPoint := "CU2~PN~585A1_ModuleAccessPoint", AxisID := "CU2_ID_1_585A1", TokenChain := "TOKENCHAIN_CU2", Simulation :=, Alarm := #Alarm.CU_585A1, Warning := #Warning.CU_585A1, Diag := #Diag.CU_585A1, AlarmPresence =>, WarningPresence =>)
   END_RUNG
   RUNG wire#powerrail
      Contact( #CU_585A1.WarningPresence )
      wire#w1
      { S7_Templates := "SrcType := UInt" } EQ_Contact(in1 := #Diag.CU_585A1.Drive_Message, in2 := #MSG_A1073_POWER_ON_REQ_BACKUP_COPY)
      wire#w2
      R_Coil( #Warning.CU_585A1.CUWarning )
   END_RUNG
   RUNG wire#w1
      { S7_Templates := "SrcType := UInt" } EQ_Contact(in1 := #Diag.CU_585A1.Drive_Message, in2 := #MSG_A13030_TRIAL_LICENSE_ACTIVATE)
   END_RUNG wire#w2
   // the same network as SCL:
   #CU_585A1(Rst := #Ctrl.RstAlarms,   // "SinamicsCU_Modulblock"
             Tel393_HWID := "HW_Const_Values".CU2_PN_585A1_SIEMENS_telegram_393,
             AccessPoint := "CU2~PN~585A1_ModuleAccessPoint",
             AxisID := "CU2_ID_1_585A1",
             TokenChain := "TOKENCHAIN_CU2",
             Alarm := #Alarm.CU_585A1,
             Warning := #Warning.CU_585A1,
             Diag := #Diag.CU_585A1);
   IF #CU_585A1.WarningPresence AND ((#Diag.CU_585A1.Drive_Message = #MSG_A1073_POWER_ON_REQ_BACKUP_COPY) OR (#Diag.CU_585A1.Drive_Message = #MSG_A13030_TRIAL_LICENSE_ACTIVATE)) THEN
       #Warning.CU_585A1.CUWarning := FALSE;
   END_IF;
END_REGION

REGION Network 16: CU 590A1
   // Bypass message "POWER ON REQUIRED FOR COPY ON MEMORY CARD"
   RUNG wire#powerrail
      #CU_590A1(Rst := #Ctrl.RstAlarms, Tel393_HWID := "CU3~PROFINET_interface~590A1_SIEMENS_telegram_393", AccessPoint := "CU3~PROFINET_interface~590A1_ModuleAccessPoint", AxisID := "CU3_ID_1_590A1", TokenChain := "TOKENCHAIN_CU3", Simulation :=, Alarm := #Alarm.CU_590A1, Warning := #Warning.CU_590A1, Diag := #Diag.CU_590A1, AlarmPresence =>, WarningPresence =>)
   END_RUNG
   RUNG wire#powerrail
      Contact( #CU_590A1.WarningPresence )
      wire#w1
      { S7_Templates := "SrcType := UInt" } EQ_Contact(in1 := #Diag.CU_590A1.Drive_Message, in2 := #MSG_A1073_POWER_ON_REQ_BACKUP_COPY)
      wire#w2
      R_Coil( #Warning.CU_590A1.CUWarning )
   END_RUNG
   RUNG wire#w1
      { S7_Templates := "SrcType := UInt" } EQ_Contact(in1 := #Diag.CU_590A1.Drive_Message, in2 := #MSG_A13030_TRIAL_LICENSE_ACTIVATE)
   END_RUNG wire#w2
   // the same network as SCL:
   #CU_590A1(Rst := #Ctrl.RstAlarms,   // "SinamicsCU_Modulblock"
             Tel393_HWID := "CU3~PROFINET_interface~590A1_SIEMENS_telegram_393",
             AccessPoint := "CU3~PROFINET_interface~590A1_ModuleAccessPoint",
             AxisID := "CU3_ID_1_590A1",
             TokenChain := "TOKENCHAIN_CU3",
             Alarm := #Alarm.CU_590A1,
             Warning := #Warning.CU_590A1,
             Diag := #Diag.CU_590A1);
   IF #CU_590A1.WarningPresence AND ((#Diag.CU_590A1.Drive_Message = #MSG_A1073_POWER_ON_REQ_BACKUP_COPY) OR (#Diag.CU_590A1.Drive_Message = #MSG_A13030_TRIAL_LICENSE_ACTIVATE)) THEN
       #Warning.CU_590A1.CUWarning := FALSE;
   END_IF;
END_REGION

REGION Network 17: CU 595A1
   // Bypass message "POWER ON REQUIRED FOR COPY ON MEMORY CARD"
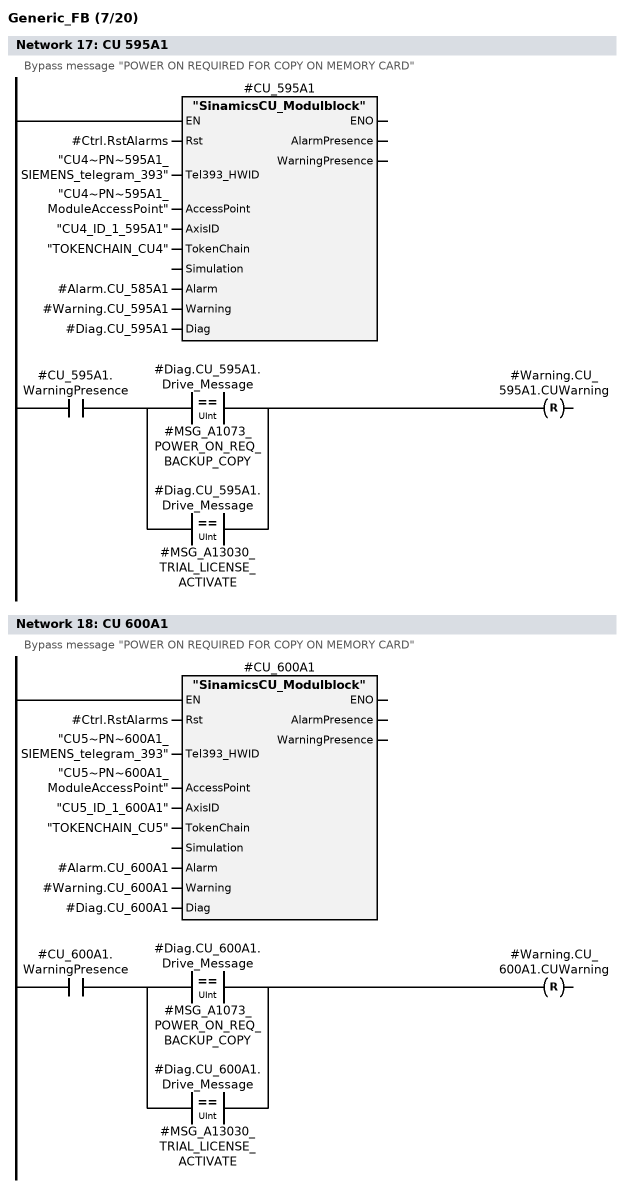
   RUNG wire#powerrail
      #CU_595A1(Rst := #Ctrl.RstAlarms, Tel393_HWID := "CU4~PN~595A1_SIEMENS_telegram_393", AccessPoint := "CU4~PN~595A1_ModuleAccessPoint", AxisID := "CU4_ID_1_595A1", TokenChain := "TOKENCHAIN_CU4", Simulation :=, Alarm := #Alarm.CU_585A1, Warning := #Warning.CU_595A1, Diag := #Diag.CU_595A1, AlarmPresence =>, WarningPresence =>)
   END_RUNG
   RUNG wire#powerrail
      Contact( #CU_595A1.WarningPresence )
      wire#w1
      { S7_Templates := "SrcType := UInt" } EQ_Contact(in1 := #Diag.CU_595A1.Drive_Message, in2 := #MSG_A1073_POWER_ON_REQ_BACKUP_COPY)
      wire#w2
      R_Coil( #Warning.CU_595A1.CUWarning )
   END_RUNG
   RUNG wire#w1
      { S7_Templates := "SrcType := UInt" } EQ_Contact(in1 := #Diag.CU_595A1.Drive_Message, in2 := #MSG_A13030_TRIAL_LICENSE_ACTIVATE)
   END_RUNG wire#w2
   // the same network as SCL:
   #CU_595A1(Rst := #Ctrl.RstAlarms,   // "SinamicsCU_Modulblock"
             Tel393_HWID := "CU4~PN~595A1_SIEMENS_telegram_393",
             AccessPoint := "CU4~PN~595A1_ModuleAccessPoint",
             AxisID := "CU4_ID_1_595A1",
             TokenChain := "TOKENCHAIN_CU4",
             Alarm := #Alarm.CU_585A1,
             Warning := #Warning.CU_595A1,
             Diag := #Diag.CU_595A1);
   IF #CU_595A1.WarningPresence AND ((#Diag.CU_595A1.Drive_Message = #MSG_A1073_POWER_ON_REQ_BACKUP_COPY) OR (#Diag.CU_595A1.Drive_Message = #MSG_A13030_TRIAL_LICENSE_ACTIVATE)) THEN
       #Warning.CU_595A1.CUWarning := FALSE;
   END_IF;
END_REGION

REGION Network 18: CU 600A1
   // Bypass message "POWER ON REQUIRED FOR COPY ON MEMORY CARD"
   RUNG wire#powerrail
      #CU_600A1(Rst := #Ctrl.RstAlarms, Tel393_HWID := "CU5~PN~600A1_SIEMENS_telegram_393", AccessPoint := "CU5~PN~600A1_ModuleAccessPoint", AxisID := "CU5_ID_1_600A1", TokenChain := "TOKENCHAIN_CU5", Simulation :=, Alarm := #Alarm.CU_600A1, Warning := #Warning.CU_600A1, Diag := #Diag.CU_600A1, AlarmPresence =>, WarningPresence =>)
   END_RUNG
   RUNG wire#powerrail
      Contact( #CU_600A1.WarningPresence )
      wire#w1
      { S7_Templates := "SrcType := UInt" } EQ_Contact(in1 := #Diag.CU_600A1.Drive_Message, in2 := #MSG_A1073_POWER_ON_REQ_BACKUP_COPY)
      wire#w2
      R_Coil( #Warning.CU_600A1.CUWarning )
   END_RUNG
   RUNG wire#w1
      { S7_Templates := "SrcType := UInt" } EQ_Contact(in1 := #Diag.CU_600A1.Drive_Message, in2 := #MSG_A13030_TRIAL_LICENSE_ACTIVATE)
   END_RUNG wire#w2
   // the same network as SCL:
   #CU_600A1(Rst := #Ctrl.RstAlarms,   // "SinamicsCU_Modulblock"
             Tel393_HWID := "CU5~PN~600A1_SIEMENS_telegram_393",
             AccessPoint := "CU5~PN~600A1_ModuleAccessPoint",
             AxisID := "CU5_ID_1_600A1",
             TokenChain := "TOKENCHAIN_CU5",
             Alarm := #Alarm.CU_600A1,
             Warning := #Warning.CU_600A1,
             Diag := #Diag.CU_600A1);
   IF #CU_600A1.WarningPresence AND ((#Diag.CU_600A1.Drive_Message = #MSG_A1073_POWER_ON_REQ_BACKUP_COPY) OR (#Diag.CU_600A1.Drive_Message = #MSG_A13030_TRIAL_LICENSE_ACTIVATE)) THEN
       #Warning.CU_600A1.CUWarning := FALSE;
   END_IF;
END_REGION

REGION Network 19: CU 605A1
   // Bypass message "POWER ON REQUIRED FOR COPY ON MEMORY CARD"
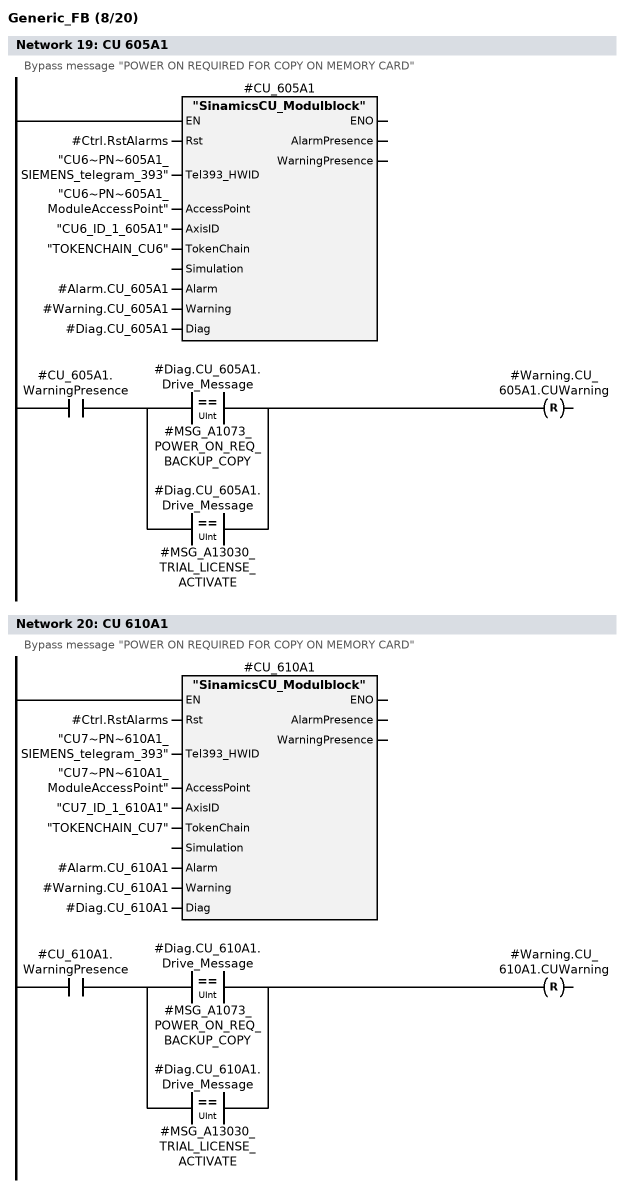
   RUNG wire#powerrail
      #CU_605A1(Rst := #Ctrl.RstAlarms, Tel393_HWID := "CU6~PN~605A1_SIEMENS_telegram_393", AccessPoint := "CU6~PN~605A1_ModuleAccessPoint", AxisID := "CU6_ID_1_605A1", TokenChain := "TOKENCHAIN_CU6", Simulation :=, Alarm := #Alarm.CU_605A1, Warning := #Warning.CU_605A1, Diag := #Diag.CU_605A1, AlarmPresence =>, WarningPresence =>)
   END_RUNG
   RUNG wire#powerrail
      Contact( #CU_605A1.WarningPresence )
      wire#w1
      { S7_Templates := "SrcType := UInt" } EQ_Contact(in1 := #Diag.CU_605A1.Drive_Message, in2 := #MSG_A1073_POWER_ON_REQ_BACKUP_COPY)
      wire#w2
      R_Coil( #Warning.CU_605A1.CUWarning )
   END_RUNG
   RUNG wire#w1
      { S7_Templates := "SrcType := UInt" } EQ_Contact(in1 := #Diag.CU_605A1.Drive_Message, in2 := #MSG_A13030_TRIAL_LICENSE_ACTIVATE)
   END_RUNG wire#w2
   // the same network as SCL:
   #CU_605A1(Rst := #Ctrl.RstAlarms,   // "SinamicsCU_Modulblock"
             Tel393_HWID := "CU6~PN~605A1_SIEMENS_telegram_393",
             AccessPoint := "CU6~PN~605A1_ModuleAccessPoint",
             AxisID := "CU6_ID_1_605A1",
             TokenChain := "TOKENCHAIN_CU6",
             Alarm := #Alarm.CU_605A1,
             Warning := #Warning.CU_605A1,
             Diag := #Diag.CU_605A1);
   IF #CU_605A1.WarningPresence AND ((#Diag.CU_605A1.Drive_Message = #MSG_A1073_POWER_ON_REQ_BACKUP_COPY) OR (#Diag.CU_605A1.Drive_Message = #MSG_A13030_TRIAL_LICENSE_ACTIVATE)) THEN
       #Warning.CU_605A1.CUWarning := FALSE;
   END_IF;
END_REGION

REGION Network 20: CU 610A1
   // Bypass message "POWER ON REQUIRED FOR COPY ON MEMORY CARD"
   RUNG wire#powerrail
      #CU_610A1(Rst := #Ctrl.RstAlarms, Tel393_HWID := "CU7~PN~610A1_SIEMENS_telegram_393", AccessPoint := "CU7~PN~610A1_ModuleAccessPoint", AxisID := "CU7_ID_1_610A1", TokenChain := "TOKENCHAIN_CU7", Simulation :=, Alarm := #Alarm.CU_610A1, Warning := #Warning.CU_610A1, Diag := #Diag.CU_610A1, AlarmPresence =>, WarningPresence =>)
   END_RUNG
   RUNG wire#powerrail
      Contact( #CU_610A1.WarningPresence )
      wire#w1
      { S7_Templates := "SrcType := UInt" } EQ_Contact(in1 := #Diag.CU_610A1.Drive_Message, in2 := #MSG_A1073_POWER_ON_REQ_BACKUP_COPY)
      wire#w2
      R_Coil( #Warning.CU_610A1.CUWarning )
   END_RUNG
   RUNG wire#w1
      { S7_Templates := "SrcType := UInt" } EQ_Contact(in1 := #Diag.CU_610A1.Drive_Message, in2 := #MSG_A13030_TRIAL_LICENSE_ACTIVATE)
   END_RUNG wire#w2
   // the same network as SCL:
   #CU_610A1(Rst := #Ctrl.RstAlarms,   // "SinamicsCU_Modulblock"
             Tel393_HWID := "CU7~PN~610A1_SIEMENS_telegram_393",
             AccessPoint := "CU7~PN~610A1_ModuleAccessPoint",
             AxisID := "CU7_ID_1_610A1",
             TokenChain := "TOKENCHAIN_CU7",
             Alarm := #Alarm.CU_610A1,
             Warning := #Warning.CU_610A1,
             Diag := #Diag.CU_610A1);
   IF #CU_610A1.WarningPresence AND ((#Diag.CU_610A1.Drive_Message = #MSG_A1073_POWER_ON_REQ_BACKUP_COPY) OR (#Diag.CU_610A1.Drive_Message = #MSG_A13030_TRIAL_LICENSE_ACTIVATE)) THEN
       #Warning.CU_610A1.CUWarning := FALSE;
   END_IF;
END_REGION

REGION Network 21: CU 615A1
   // Bypass message "POWER ON REQUIRED FOR COPY ON MEMORY CARD"
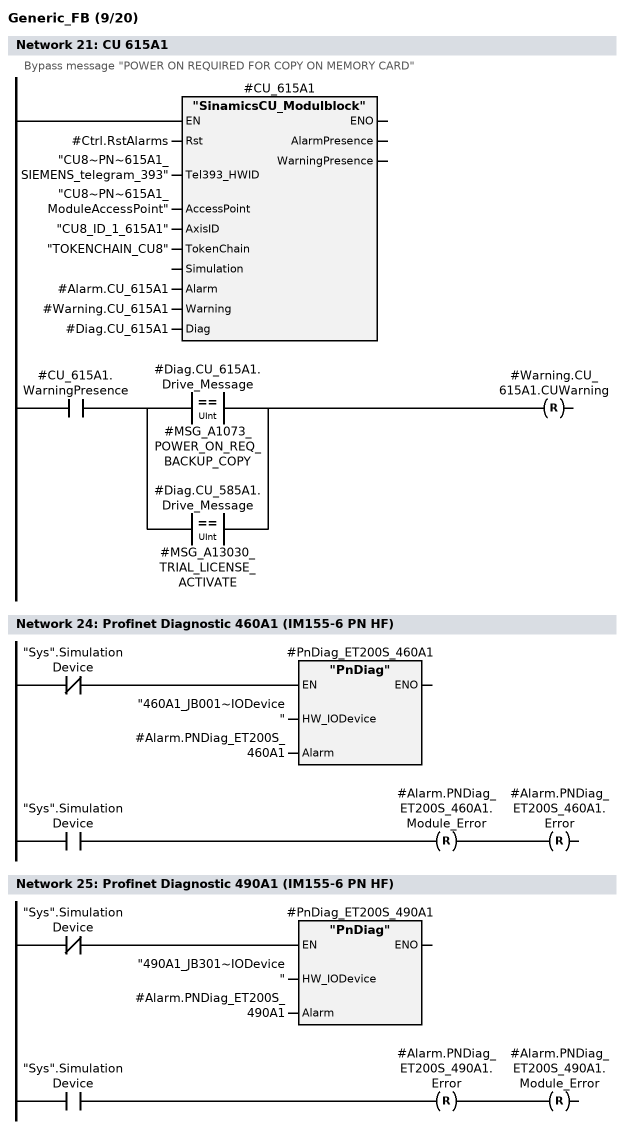
   RUNG wire#powerrail
      #CU_615A1(Rst := #Ctrl.RstAlarms, Tel393_HWID := "CU8~PN~615A1_SIEMENS_telegram_393", AccessPoint := "CU8~PN~615A1_ModuleAccessPoint", AxisID := "CU8_ID_1_615A1", TokenChain := "TOKENCHAIN_CU8", Simulation :=, Alarm := #Alarm.CU_615A1, Warning := #Warning.CU_615A1, Diag := #Diag.CU_615A1, AlarmPresence =>, WarningPresence =>)
   END_RUNG
   RUNG wire#powerrail
      Contact( #CU_615A1.WarningPresence )
      wire#w1
      { S7_Templates := "SrcType := UInt" } EQ_Contact(in1 := #Diag.CU_615A1.Drive_Message, in2 := #MSG_A1073_POWER_ON_REQ_BACKUP_COPY)
      wire#w2
      R_Coil( #Warning.CU_615A1.CUWarning )
   END_RUNG
   RUNG wire#w1
      { S7_Templates := "SrcType := UInt" } EQ_Contact(in1 := #Diag.CU_585A1.Drive_Message, in2 := #MSG_A13030_TRIAL_LICENSE_ACTIVATE)
   END_RUNG wire#w2
   // the same network as SCL:
   #CU_615A1(Rst := #Ctrl.RstAlarms,   // "SinamicsCU_Modulblock"
             Tel393_HWID := "CU8~PN~615A1_SIEMENS_telegram_393",
             AccessPoint := "CU8~PN~615A1_ModuleAccessPoint",
             AxisID := "CU8_ID_1_615A1",
             TokenChain := "TOKENCHAIN_CU8",
             Alarm := #Alarm.CU_615A1,
             Warning := #Warning.CU_615A1,
             Diag := #Diag.CU_615A1);
   IF #CU_615A1.WarningPresence AND ((#Diag.CU_615A1.Drive_Message = #MSG_A1073_POWER_ON_REQ_BACKUP_COPY) OR (#Diag.CU_585A1.Drive_Message = #MSG_A13030_TRIAL_LICENSE_ACTIVATE)) THEN
       #Warning.CU_615A1.CUWarning := FALSE;
   END_IF;
END_REGION

REGION Network 23: <<< PROFINET DIAGNOSTIC >>>
END_REGION

REGION Network 24: Profinet Diagnostic 460A1 (IM155-6 PN HF)
   RUNG wire#powerrail
      I_Contact( "Sys".SimulationDevice )
      #PnDiag_ET200S_460A1(HW_IODevice := "460A1_JB001~IODevice", Alarm := #Alarm.PNDiag_ET200S_460A1)
   END_RUNG
   RUNG wire#powerrail
      Contact( "Sys".SimulationDevice )
      R_Coil( #Alarm.PNDiag_ET200S_460A1.Module_Error )
      R_Coil( #Alarm.PNDiag_ET200S_460A1.Error )
   END_RUNG
   // the same network as SCL:
   IF NOT "Sys".SimulationDevice THEN
       #PnDiag_ET200S_460A1(HW_IODevice := "460A1_JB001~IODevice", Alarm := #Alarm.PNDiag_ET200S_460A1);   // "PnDiag"
   END_IF;
   IF "Sys".SimulationDevice THEN
       #Alarm.PNDiag_ET200S_460A1.Module_Error := FALSE;
       #Alarm.PNDiag_ET200S_460A1.Error := FALSE;
   END_IF;
END_REGION

REGION Network 25: Profinet Diagnostic 490A1 (IM155-6 PN HF)
   RUNG wire#powerrail
      I_Contact( "Sys".SimulationDevice )
      #PnDiag_ET200S_490A1(HW_IODevice := "490A1_JB301~IODevice", Alarm := #Alarm.PNDiag_ET200S_490A1)
   END_RUNG
   RUNG wire#powerrail
      Contact( "Sys".SimulationDevice )
      R_Coil( #Alarm.PNDiag_ET200S_490A1.Error )
      R_Coil( #Alarm.PNDiag_ET200S_490A1.Module_Error )
   END_RUNG
   // the same network as SCL:
   IF NOT "Sys".SimulationDevice THEN
       #PnDiag_ET200S_490A1(HW_IODevice := "490A1_JB301~IODevice", Alarm := #Alarm.PNDiag_ET200S_490A1);   // "PnDiag"
   END_IF;
   IF "Sys".SimulationDevice THEN
       #Alarm.PNDiag_ET200S_490A1.Error := FALSE;
       #Alarm.PNDiag_ET200S_490A1.Module_Error := FALSE;
   END_IF;
END_REGION

REGION Network 26: Profinet Diagnostic 510A1 (IM155-6 PN HF)
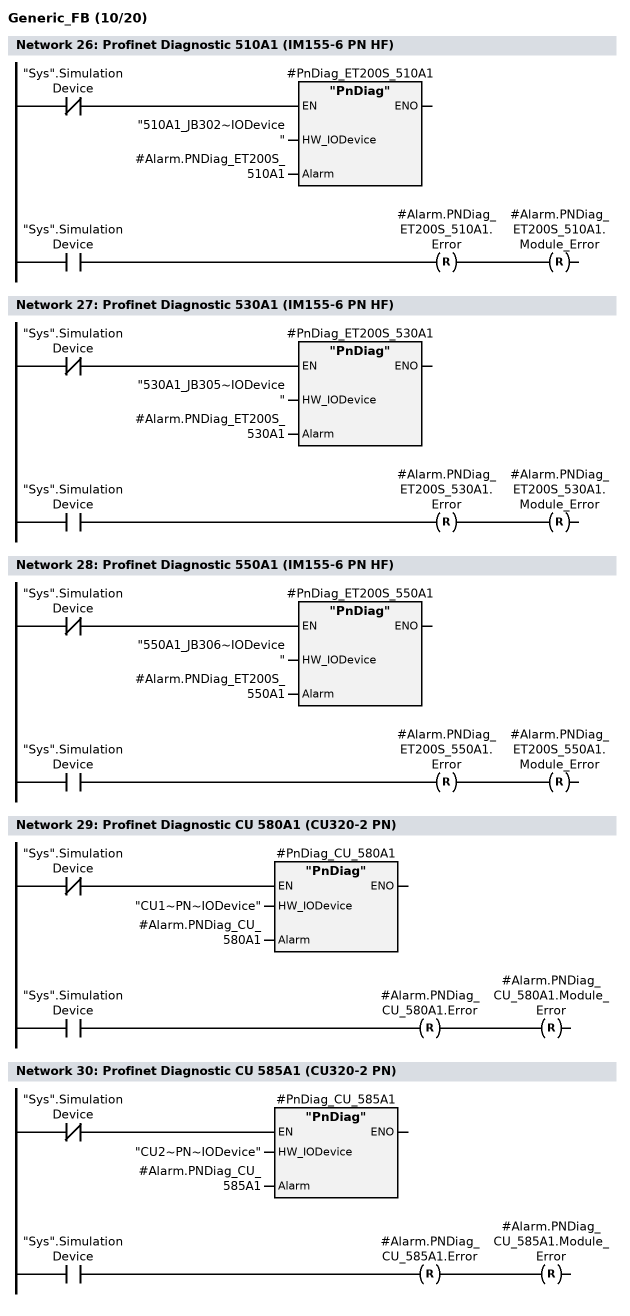
   RUNG wire#powerrail
      I_Contact( "Sys".SimulationDevice )
      #PnDiag_ET200S_510A1(HW_IODevice := "510A1_JB302~IODevice", Alarm := #Alarm.PNDiag_ET200S_510A1)
   END_RUNG
   RUNG wire#powerrail
      Contact( "Sys".SimulationDevice )
      R_Coil( #Alarm.PNDiag_ET200S_510A1.Error )
      R_Coil( #Alarm.PNDiag_ET200S_510A1.Module_Error )
   END_RUNG
   // the same network as SCL:
   IF NOT "Sys".SimulationDevice THEN
       #PnDiag_ET200S_510A1(HW_IODevice := "510A1_JB302~IODevice", Alarm := #Alarm.PNDiag_ET200S_510A1);   // "PnDiag"
   END_IF;
   IF "Sys".SimulationDevice THEN
       #Alarm.PNDiag_ET200S_510A1.Error := FALSE;
       #Alarm.PNDiag_ET200S_510A1.Module_Error := FALSE;
   END_IF;
END_REGION

REGION Network 27: Profinet Diagnostic 530A1 (IM155-6 PN HF)
   RUNG wire#powerrail
      I_Contact( "Sys".SimulationDevice )
      #PnDiag_ET200S_530A1(HW_IODevice := "530A1_JB305~IODevice", Alarm := #Alarm.PNDiag_ET200S_530A1)
   END_RUNG
   RUNG wire#powerrail
      Contact( "Sys".SimulationDevice )
      R_Coil( #Alarm.PNDiag_ET200S_530A1.Error )
      R_Coil( #Alarm.PNDiag_ET200S_530A1.Module_Error )
   END_RUNG
   // the same network as SCL:
   IF NOT "Sys".SimulationDevice THEN
       #PnDiag_ET200S_530A1(HW_IODevice := "530A1_JB305~IODevice", Alarm := #Alarm.PNDiag_ET200S_530A1);   // "PnDiag"
   END_IF;
   IF "Sys".SimulationDevice THEN
       #Alarm.PNDiag_ET200S_530A1.Error := FALSE;
       #Alarm.PNDiag_ET200S_530A1.Module_Error := FALSE;
   END_IF;
END_REGION

REGION Network 28: Profinet Diagnostic 550A1 (IM155-6 PN HF)
   RUNG wire#powerrail
      I_Contact( "Sys".SimulationDevice )
      #PnDiag_ET200S_550A1(HW_IODevice := "550A1_JB306~IODevice", Alarm := #Alarm.PNDiag_ET200S_550A1)
   END_RUNG
   RUNG wire#powerrail
      Contact( "Sys".SimulationDevice )
      R_Coil( #Alarm.PNDiag_ET200S_550A1.Error )
      R_Coil( #Alarm.PNDiag_ET200S_550A1.Module_Error )
   END_RUNG
   // the same network as SCL:
   IF NOT "Sys".SimulationDevice THEN
       #PnDiag_ET200S_550A1(HW_IODevice := "550A1_JB306~IODevice", Alarm := #Alarm.PNDiag_ET200S_550A1);   // "PnDiag"
   END_IF;
   IF "Sys".SimulationDevice THEN
       #Alarm.PNDiag_ET200S_550A1.Error := FALSE;
       #Alarm.PNDiag_ET200S_550A1.Module_Error := FALSE;
   END_IF;
END_REGION

REGION Network 29: Profinet Diagnostic CU 580A1 (CU320-2 PN)
   RUNG wire#powerrail
      I_Contact( "Sys".SimulationDevice )
      #PnDiag_CU_580A1(HW_IODevice := "CU1~PN~IODevice", Alarm := #Alarm.PNDiag_CU_580A1)
   END_RUNG
   RUNG wire#powerrail
      Contact( "Sys".SimulationDevice )
      R_Coil( #Alarm.PNDiag_CU_580A1.Error )
      R_Coil( #Alarm.PNDiag_CU_580A1.Module_Error )
   END_RUNG
   // the same network as SCL:
   IF NOT "Sys".SimulationDevice THEN
       #PnDiag_CU_580A1(HW_IODevice := "CU1~PN~IODevice", Alarm := #Alarm.PNDiag_CU_580A1);   // "PnDiag"
   END_IF;
   IF "Sys".SimulationDevice THEN
       #Alarm.PNDiag_CU_580A1.Error := FALSE;
       #Alarm.PNDiag_CU_580A1.Module_Error := FALSE;
   END_IF;
END_REGION

REGION Network 30: Profinet Diagnostic CU 585A1 (CU320-2 PN)
   RUNG wire#powerrail
      I_Contact( "Sys".SimulationDevice )
      #PnDiag_CU_585A1(HW_IODevice := "CU2~PN~IODevice", Alarm := #Alarm.PNDiag_CU_585A1)
   END_RUNG
   RUNG wire#powerrail
      Contact( "Sys".SimulationDevice )
      R_Coil( #Alarm.PNDiag_CU_585A1.Error )
      R_Coil( #Alarm.PNDiag_CU_585A1.Module_Error )
   END_RUNG
   // the same network as SCL:
   IF NOT "Sys".SimulationDevice THEN
       #PnDiag_CU_585A1(HW_IODevice := "CU2~PN~IODevice", Alarm := #Alarm.PNDiag_CU_585A1);   // "PnDiag"
   END_IF;
   IF "Sys".SimulationDevice THEN
       #Alarm.PNDiag_CU_585A1.Error := FALSE;
       #Alarm.PNDiag_CU_585A1.Module_Error := FALSE;
   END_IF;
END_REGION

REGION Network 31: Profinet Diagnostic CU 590A1 (CU320-2 PN)
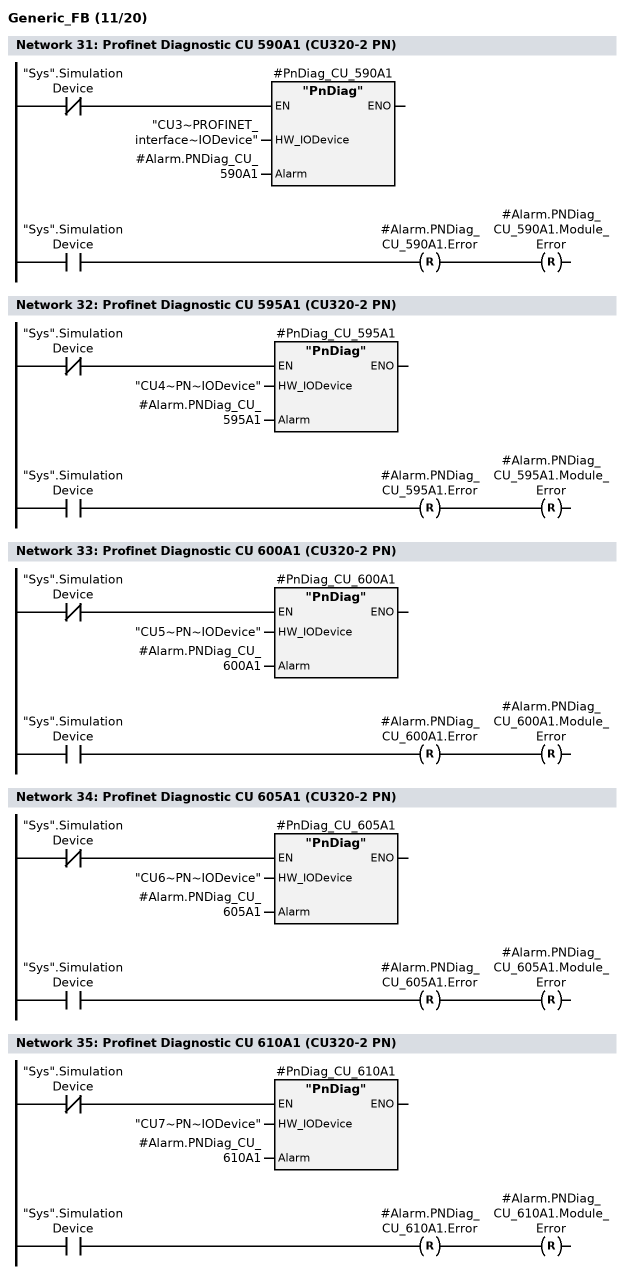
   RUNG wire#powerrail
      I_Contact( "Sys".SimulationDevice )
      #PnDiag_CU_590A1(HW_IODevice := "CU3~PROFINET_interface~IODevice", Alarm := #Alarm.PNDiag_CU_590A1)
   END_RUNG
   RUNG wire#powerrail
      Contact( "Sys".SimulationDevice )
      R_Coil( #Alarm.PNDiag_CU_590A1.Error )
      R_Coil( #Alarm.PNDiag_CU_590A1.Module_Error )
   END_RUNG
   // the same network as SCL:
   IF NOT "Sys".SimulationDevice THEN
       #PnDiag_CU_590A1(HW_IODevice := "CU3~PROFINET_interface~IODevice", Alarm := #Alarm.PNDiag_CU_590A1);   // "PnDiag"
   END_IF;
   IF "Sys".SimulationDevice THEN
       #Alarm.PNDiag_CU_590A1.Error := FALSE;
       #Alarm.PNDiag_CU_590A1.Module_Error := FALSE;
   END_IF;
END_REGION

REGION Network 32: Profinet Diagnostic CU 595A1 (CU320-2 PN)
   RUNG wire#powerrail
      I_Contact( "Sys".SimulationDevice )
      #PnDiag_CU_595A1(HW_IODevice := "CU4~PN~IODevice", Alarm := #Alarm.PNDiag_CU_595A1)
   END_RUNG
   RUNG wire#powerrail
      Contact( "Sys".SimulationDevice )
      R_Coil( #Alarm.PNDiag_CU_595A1.Error )
      R_Coil( #Alarm.PNDiag_CU_595A1.Module_Error )
   END_RUNG
   // the same network as SCL:
   IF NOT "Sys".SimulationDevice THEN
       #PnDiag_CU_595A1(HW_IODevice := "CU4~PN~IODevice", Alarm := #Alarm.PNDiag_CU_595A1);   // "PnDiag"
   END_IF;
   IF "Sys".SimulationDevice THEN
       #Alarm.PNDiag_CU_595A1.Error := FALSE;
       #Alarm.PNDiag_CU_595A1.Module_Error := FALSE;
   END_IF;
END_REGION

REGION Network 33: Profinet Diagnostic CU 600A1 (CU320-2 PN)
   RUNG wire#powerrail
      I_Contact( "Sys".SimulationDevice )
      #PnDiag_CU_600A1(HW_IODevice := "CU5~PN~IODevice", Alarm := #Alarm.PNDiag_CU_600A1)
   END_RUNG
   RUNG wire#powerrail
      Contact( "Sys".SimulationDevice )
      R_Coil( #Alarm.PNDiag_CU_600A1.Error )
      R_Coil( #Alarm.PNDiag_CU_600A1.Module_Error )
   END_RUNG
   // the same network as SCL:
   IF NOT "Sys".SimulationDevice THEN
       #PnDiag_CU_600A1(HW_IODevice := "CU5~PN~IODevice", Alarm := #Alarm.PNDiag_CU_600A1);   // "PnDiag"
   END_IF;
   IF "Sys".SimulationDevice THEN
       #Alarm.PNDiag_CU_600A1.Error := FALSE;
       #Alarm.PNDiag_CU_600A1.Module_Error := FALSE;
   END_IF;
END_REGION

REGION Network 34: Profinet Diagnostic CU 605A1 (CU320-2 PN)
   RUNG wire#powerrail
      I_Contact( "Sys".SimulationDevice )
      #PnDiag_CU_605A1(HW_IODevice := "CU6~PN~IODevice", Alarm := #Alarm.PNDiag_CU_605A1)
   END_RUNG
   RUNG wire#powerrail
      Contact( "Sys".SimulationDevice )
      R_Coil( #Alarm.PNDiag_CU_605A1.Error )
      R_Coil( #Alarm.PNDiag_CU_605A1.Module_Error )
   END_RUNG
   // the same network as SCL:
   IF NOT "Sys".SimulationDevice THEN
       #PnDiag_CU_605A1(HW_IODevice := "CU6~PN~IODevice", Alarm := #Alarm.PNDiag_CU_605A1);   // "PnDiag"
   END_IF;
   IF "Sys".SimulationDevice THEN
       #Alarm.PNDiag_CU_605A1.Error := FALSE;
       #Alarm.PNDiag_CU_605A1.Module_Error := FALSE;
   END_IF;
END_REGION

REGION Network 35: Profinet Diagnostic CU 610A1 (CU320-2 PN)
   RUNG wire#powerrail
      I_Contact( "Sys".SimulationDevice )
      #PnDiag_CU_610A1(HW_IODevice := "CU7~PN~IODevice", Alarm := #Alarm.PNDiag_CU_610A1)
   END_RUNG
   RUNG wire#powerrail
      Contact( "Sys".SimulationDevice )
      R_Coil( #Alarm.PNDiag_CU_610A1.Error )
      R_Coil( #Alarm.PNDiag_CU_610A1.Module_Error )
   END_RUNG
   // the same network as SCL:
   IF NOT "Sys".SimulationDevice THEN
       #PnDiag_CU_610A1(HW_IODevice := "CU7~PN~IODevice", Alarm := #Alarm.PNDiag_CU_610A1);   // "PnDiag"
   END_IF;
   IF "Sys".SimulationDevice THEN
       #Alarm.PNDiag_CU_610A1.Error := FALSE;
       #Alarm.PNDiag_CU_610A1.Module_Error := FALSE;
   END_IF;
END_REGION

REGION Network 36: Profinet Diagnostic CU 615A1 (CU320-2 PN)
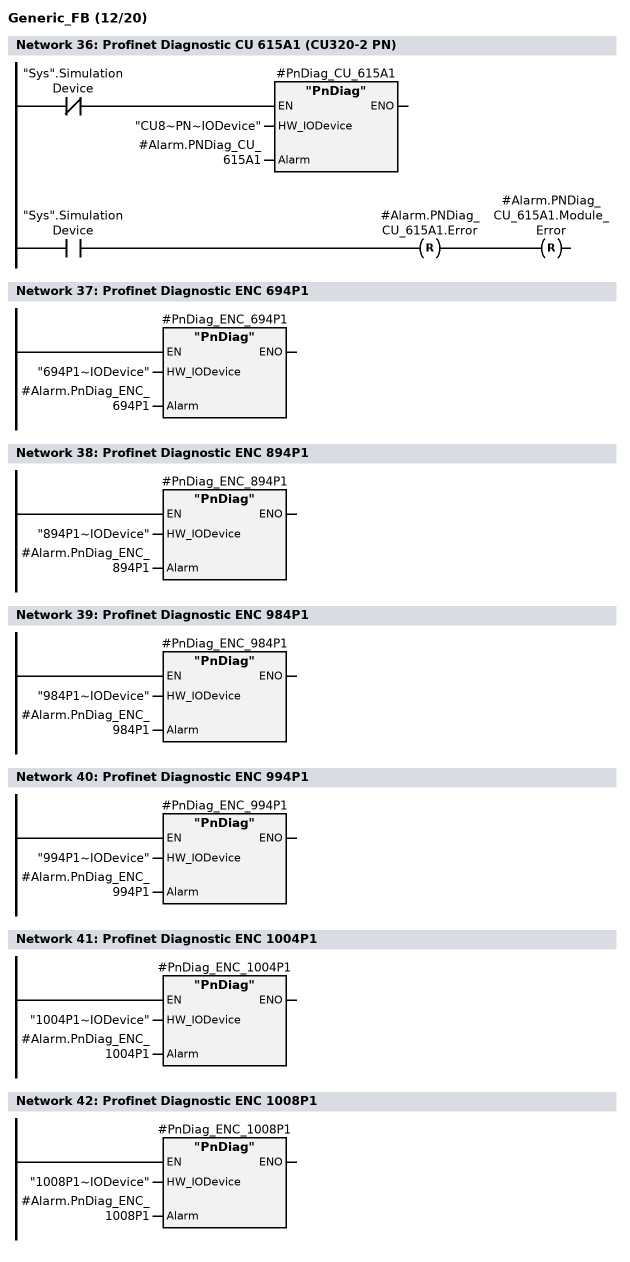
   RUNG wire#powerrail
      I_Contact( "Sys".SimulationDevice )
      #PnDiag_CU_615A1(HW_IODevice := "CU8~PN~IODevice", Alarm := #Alarm.PNDiag_CU_615A1)
   END_RUNG
   RUNG wire#powerrail
      Contact( "Sys".SimulationDevice )
      R_Coil( #Alarm.PNDiag_CU_615A1.Error )
      R_Coil( #Alarm.PNDiag_CU_615A1.Module_Error )
   END_RUNG
   // the same network as SCL:
   IF NOT "Sys".SimulationDevice THEN
       #PnDiag_CU_615A1(HW_IODevice := "CU8~PN~IODevice", Alarm := #Alarm.PNDiag_CU_615A1);   // "PnDiag"
   END_IF;
   IF "Sys".SimulationDevice THEN
       #Alarm.PNDiag_CU_615A1.Error := FALSE;
       #Alarm.PNDiag_CU_615A1.Module_Error := FALSE;
   END_IF;
END_REGION

REGION Network 37: Profinet Diagnostic ENC 694P1
   RUNG wire#powerrail
      #PnDiag_ENC_694P1(HW_IODevice := "694P1~IODevice", Alarm := #Alarm.PnDiag_ENC_694P1)
   END_RUNG
   // the same network as SCL:
   #PnDiag_ENC_694P1(HW_IODevice := "694P1~IODevice", Alarm := #Alarm.PnDiag_ENC_694P1);   // "PnDiag"
END_REGION

REGION Network 38: Profinet Diagnostic ENC 894P1
   RUNG wire#powerrail
      #PnDiag_ENC_894P1(HW_IODevice := "894P1~IODevice", Alarm := #Alarm.PnDiag_ENC_894P1)
   END_RUNG
   // the same network as SCL:
   #PnDiag_ENC_894P1(HW_IODevice := "894P1~IODevice", Alarm := #Alarm.PnDiag_ENC_894P1);   // "PnDiag"
END_REGION

REGION Network 39: Profinet Diagnostic ENC 984P1
   RUNG wire#powerrail
      #PnDiag_ENC_984P1(HW_IODevice := "984P1~IODevice", Alarm := #Alarm.PnDiag_ENC_984P1)
   END_RUNG
   // the same network as SCL:
   #PnDiag_ENC_984P1(HW_IODevice := "984P1~IODevice", Alarm := #Alarm.PnDiag_ENC_984P1);   // "PnDiag"
END_REGION

REGION Network 40: Profinet Diagnostic ENC 994P1
   RUNG wire#powerrail
      #PnDiag_ENC_994P1(HW_IODevice := "994P1~IODevice", Alarm := #Alarm.PnDiag_ENC_994P1)
   END_RUNG
   // the same network as SCL:
   #PnDiag_ENC_994P1(HW_IODevice := "994P1~IODevice", Alarm := #Alarm.PnDiag_ENC_994P1);   // "PnDiag"
END_REGION

REGION Network 41: Profinet Diagnostic ENC 1004P1
   RUNG wire#powerrail
      #PnDiag_ENC_1004P1(HW_IODevice := "1004P1~IODevice", Alarm := #Alarm.PnDiag_ENC_1004P1)
   END_RUNG
   // the same network as SCL:
   #PnDiag_ENC_1004P1(HW_IODevice := "1004P1~IODevice", Alarm := #Alarm.PnDiag_ENC_1004P1);   // "PnDiag"
END_REGION

REGION Network 42: Profinet Diagnostic ENC 1008P1
   RUNG wire#powerrail
      #PnDiag_ENC_1008P1(HW_IODevice := "1008P1~IODevice", Alarm := #Alarm.PnDiag_ENC_1008P1)
   END_RUNG
   // the same network as SCL:
   #PnDiag_ENC_1008P1(HW_IODevice := "1008P1~IODevice", Alarm := #Alarm.PnDiag_ENC_1008P1);   // "PnDiag"
END_REGION

REGION Network 43: Profinet Diagnostic ENC 1034P1
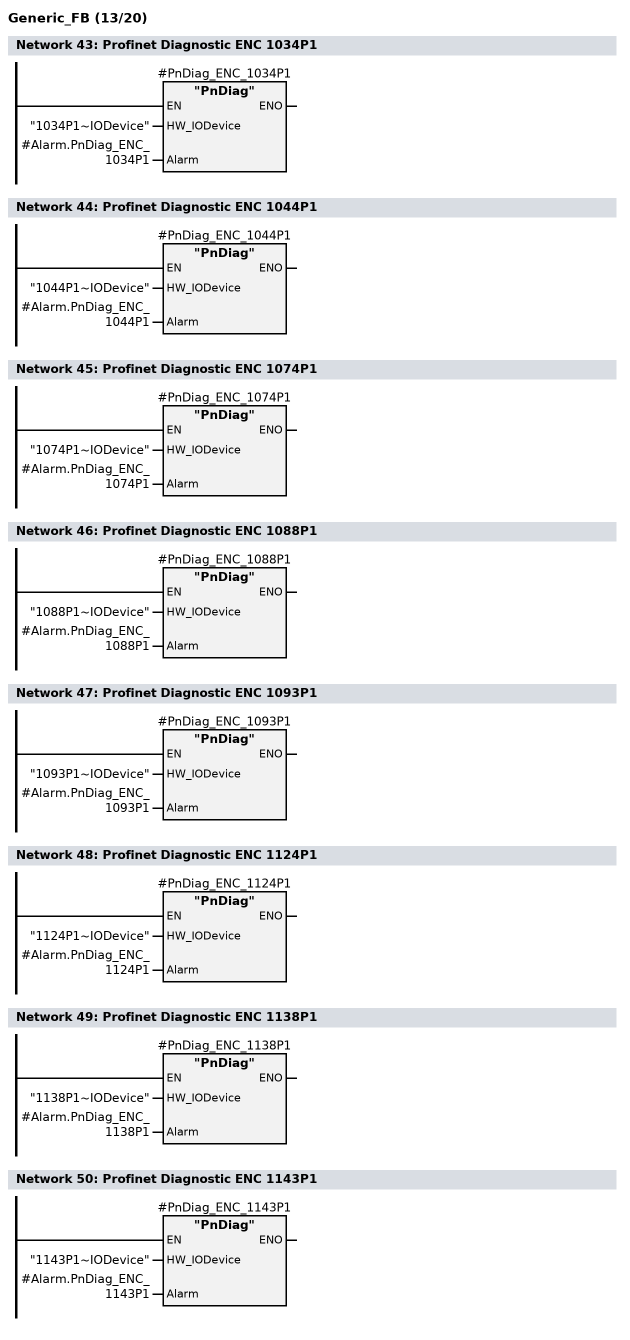
   RUNG wire#powerrail
      #PnDiag_ENC_1034P1(HW_IODevice := "1034P1~IODevice", Alarm := #Alarm.PnDiag_ENC_1034P1)
   END_RUNG
   // the same network as SCL:
   #PnDiag_ENC_1034P1(HW_IODevice := "1034P1~IODevice", Alarm := #Alarm.PnDiag_ENC_1034P1);   // "PnDiag"
END_REGION

REGION Network 44: Profinet Diagnostic ENC 1044P1
   RUNG wire#powerrail
      #PnDiag_ENC_1044P1(HW_IODevice := "1044P1~IODevice", Alarm := #Alarm.PnDiag_ENC_1044P1)
   END_RUNG
   // the same network as SCL:
   #PnDiag_ENC_1044P1(HW_IODevice := "1044P1~IODevice", Alarm := #Alarm.PnDiag_ENC_1044P1);   // "PnDiag"
END_REGION

REGION Network 45: Profinet Diagnostic ENC 1074P1
   RUNG wire#powerrail
      #PnDiag_ENC_1074P1(HW_IODevice := "1074P1~IODevice", Alarm := #Alarm.PnDiag_ENC_1074P1)
   END_RUNG
   // the same network as SCL:
   #PnDiag_ENC_1074P1(HW_IODevice := "1074P1~IODevice", Alarm := #Alarm.PnDiag_ENC_1074P1);   // "PnDiag"
END_REGION

REGION Network 46: Profinet Diagnostic ENC 1088P1
   RUNG wire#powerrail
      #PnDiag_ENC_1088P1(HW_IODevice := "1088P1~IODevice", Alarm := #Alarm.PnDiag_ENC_1088P1)
   END_RUNG
   // the same network as SCL:
   #PnDiag_ENC_1088P1(HW_IODevice := "1088P1~IODevice", Alarm := #Alarm.PnDiag_ENC_1088P1);   // "PnDiag"
END_REGION

REGION Network 47: Profinet Diagnostic ENC 1093P1
   RUNG wire#powerrail
      #PnDiag_ENC_1093P1(HW_IODevice := "1093P1~IODevice", Alarm := #Alarm.PnDiag_ENC_1093P1)
   END_RUNG
   // the same network as SCL:
   #PnDiag_ENC_1093P1(HW_IODevice := "1093P1~IODevice", Alarm := #Alarm.PnDiag_ENC_1093P1);   // "PnDiag"
END_REGION

REGION Network 48: Profinet Diagnostic ENC 1124P1
   RUNG wire#powerrail
      #PnDiag_ENC_1124P1(HW_IODevice := "1124P1~IODevice", Alarm := #Alarm.PnDiag_ENC_1124P1)
   END_RUNG
   // the same network as SCL:
   #PnDiag_ENC_1124P1(HW_IODevice := "1124P1~IODevice", Alarm := #Alarm.PnDiag_ENC_1124P1);   // "PnDiag"
END_REGION

REGION Network 49: Profinet Diagnostic ENC 1138P1
   RUNG wire#powerrail
      #PnDiag_ENC_1138P1(HW_IODevice := "1138P1~IODevice", Alarm := #Alarm.PnDiag_ENC_1138P1)
   END_RUNG
   // the same network as SCL:
   #PnDiag_ENC_1138P1(HW_IODevice := "1138P1~IODevice", Alarm := #Alarm.PnDiag_ENC_1138P1);   // "PnDiag"
END_REGION

REGION Network 50: Profinet Diagnostic ENC 1143P1
   RUNG wire#powerrail
      #PnDiag_ENC_1143P1(HW_IODevice := "1143P1~IODevice", Alarm := #Alarm.PnDiag_ENC_1143P1)
   END_RUNG
   // the same network as SCL:
   #PnDiag_ENC_1143P1(HW_IODevice := "1143P1~IODevice", Alarm := #Alarm.PnDiag_ENC_1143P1);   // "PnDiag"
END_REGION

REGION Network 51: Profinet Diagnostic ENC 1844P1
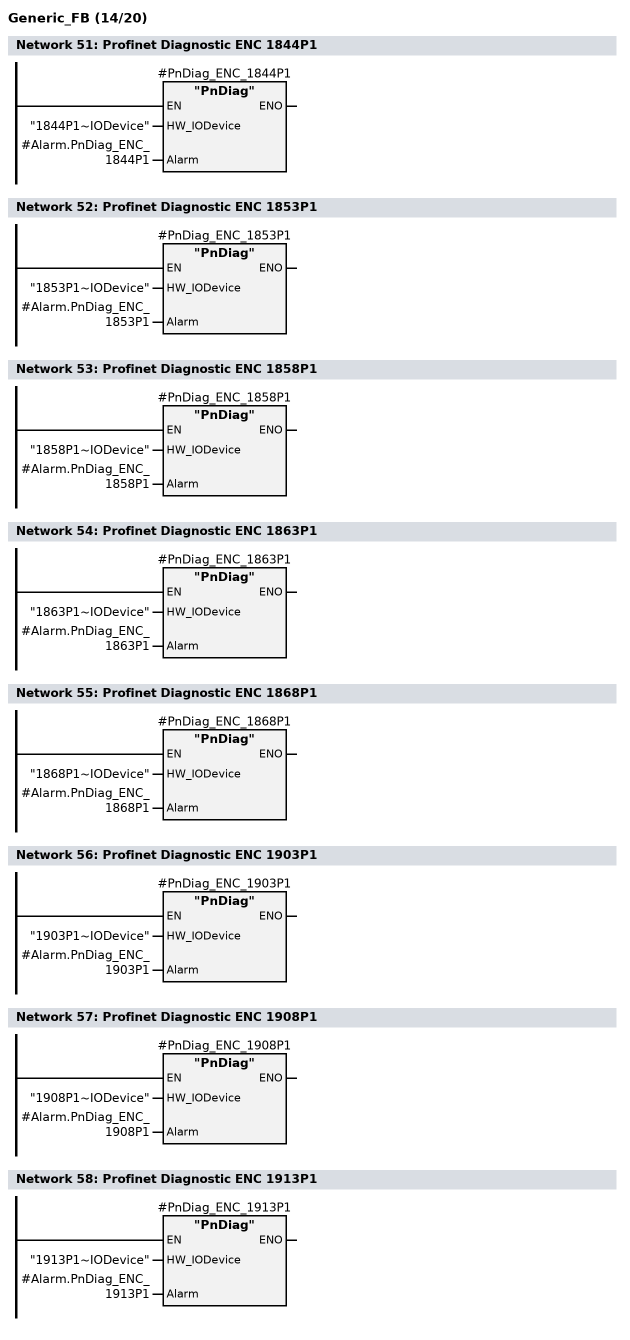
   RUNG wire#powerrail
      #PnDiag_ENC_1844P1(HW_IODevice := "1844P1~IODevice", Alarm := #Alarm.PnDiag_ENC_1844P1)
   END_RUNG
   // the same network as SCL:
   #PnDiag_ENC_1844P1(HW_IODevice := "1844P1~IODevice", Alarm := #Alarm.PnDiag_ENC_1844P1);   // "PnDiag"
END_REGION

REGION Network 52: Profinet Diagnostic ENC 1853P1
   RUNG wire#powerrail
      #PnDiag_ENC_1853P1(HW_IODevice := "1853P1~IODevice", Alarm := #Alarm.PnDiag_ENC_1853P1)
   END_RUNG
   // the same network as SCL:
   #PnDiag_ENC_1853P1(HW_IODevice := "1853P1~IODevice", Alarm := #Alarm.PnDiag_ENC_1853P1);   // "PnDiag"
END_REGION

REGION Network 53: Profinet Diagnostic ENC 1858P1
   RUNG wire#powerrail
      #PnDiag_ENC_1858P1(HW_IODevice := "1858P1~IODevice", Alarm := #Alarm.PnDiag_ENC_1858P1)
   END_RUNG
   // the same network as SCL:
   #PnDiag_ENC_1858P1(HW_IODevice := "1858P1~IODevice", Alarm := #Alarm.PnDiag_ENC_1858P1);   // "PnDiag"
END_REGION

REGION Network 54: Profinet Diagnostic ENC 1863P1
   RUNG wire#powerrail
      #PnDiag_ENC_1863P1(HW_IODevice := "1863P1~IODevice", Alarm := #Alarm.PnDiag_ENC_1863P1)
   END_RUNG
   // the same network as SCL:
   #PnDiag_ENC_1863P1(HW_IODevice := "1863P1~IODevice", Alarm := #Alarm.PnDiag_ENC_1863P1);   // "PnDiag"
END_REGION

REGION Network 55: Profinet Diagnostic ENC 1868P1
   RUNG wire#powerrail
      #PnDiag_ENC_1868P1(HW_IODevice := "1868P1~IODevice", Alarm := #Alarm.PnDiag_ENC_1868P1)
   END_RUNG
   // the same network as SCL:
   #PnDiag_ENC_1868P1(HW_IODevice := "1868P1~IODevice", Alarm := #Alarm.PnDiag_ENC_1868P1);   // "PnDiag"
END_REGION

REGION Network 56: Profinet Diagnostic ENC 1903P1
   RUNG wire#powerrail
      #PnDiag_ENC_1903P1(HW_IODevice := "1903P1~IODevice", Alarm := #Alarm.PnDiag_ENC_1903P1)
   END_RUNG
   // the same network as SCL:
   #PnDiag_ENC_1903P1(HW_IODevice := "1903P1~IODevice", Alarm := #Alarm.PnDiag_ENC_1903P1);   // "PnDiag"
END_REGION

REGION Network 57: Profinet Diagnostic ENC 1908P1
   RUNG wire#powerrail
      #PnDiag_ENC_1908P1(HW_IODevice := "1908P1~IODevice", Alarm := #Alarm.PnDiag_ENC_1908P1)
   END_RUNG
   // the same network as SCL:
   #PnDiag_ENC_1908P1(HW_IODevice := "1908P1~IODevice", Alarm := #Alarm.PnDiag_ENC_1908P1);   // "PnDiag"
END_REGION

REGION Network 58: Profinet Diagnostic ENC 1913P1
   RUNG wire#powerrail
      #PnDiag_ENC_1913P1(HW_IODevice := "1913P1~IODevice", Alarm := #Alarm.PnDiag_ENC_1913P1)
   END_RUNG
   // the same network as SCL:
   #PnDiag_ENC_1913P1(HW_IODevice := "1913P1~IODevice", Alarm := #Alarm.PnDiag_ENC_1913P1);   // "PnDiag"
END_REGION

REGION Network 59: Profinet Diagnostic ENC 1918P1
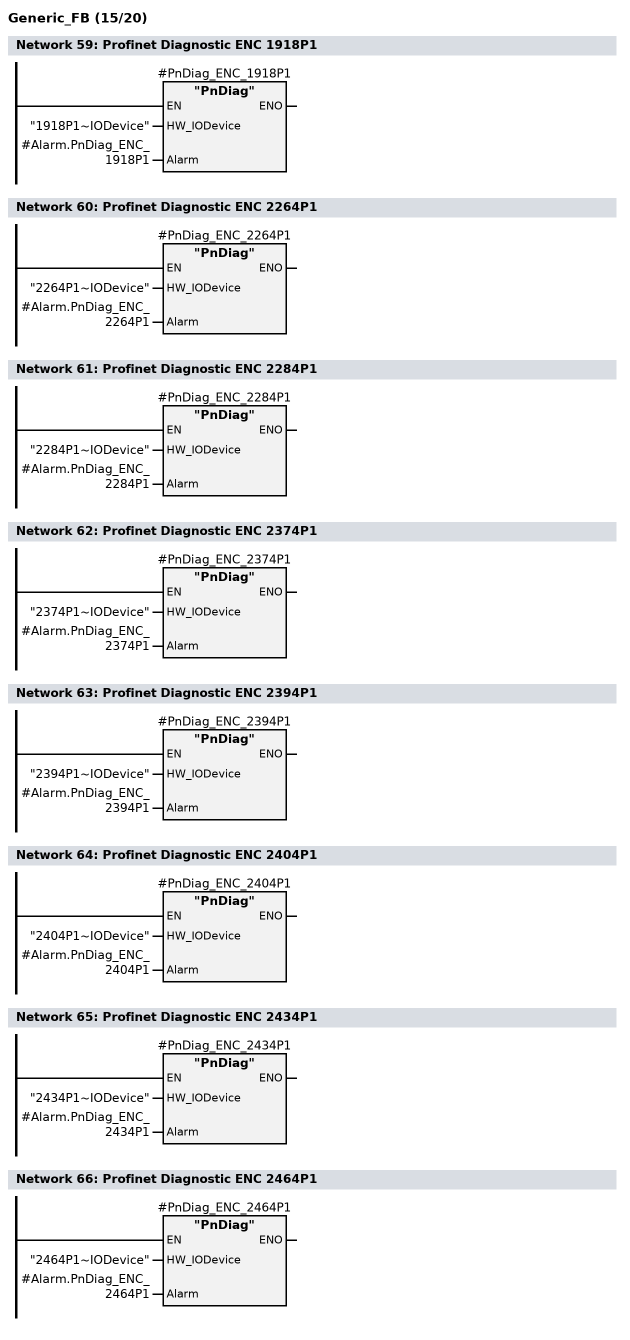
   RUNG wire#powerrail
      #PnDiag_ENC_1918P1(HW_IODevice := "1918P1~IODevice", Alarm := #Alarm.PnDiag_ENC_1918P1)
   END_RUNG
   // the same network as SCL:
   #PnDiag_ENC_1918P1(HW_IODevice := "1918P1~IODevice", Alarm := #Alarm.PnDiag_ENC_1918P1);   // "PnDiag"
END_REGION

REGION Network 60: Profinet Diagnostic ENC 2264P1
   RUNG wire#powerrail
      #PnDiag_ENC_2264P1(HW_IODevice := "2264P1~IODevice", Alarm := #Alarm.PnDiag_ENC_2264P1)
   END_RUNG
   // the same network as SCL:
   #PnDiag_ENC_2264P1(HW_IODevice := "2264P1~IODevice", Alarm := #Alarm.PnDiag_ENC_2264P1);   // "PnDiag"
END_REGION

REGION Network 61: Profinet Diagnostic ENC 2284P1
   RUNG wire#powerrail
      #PnDiag_ENC_2284P1(HW_IODevice := "2284P1~IODevice", Alarm := #Alarm.PnDiag_ENC_2284P1)
   END_RUNG
   // the same network as SCL:
   #PnDiag_ENC_2284P1(HW_IODevice := "2284P1~IODevice", Alarm := #Alarm.PnDiag_ENC_2284P1);   // "PnDiag"
END_REGION

REGION Network 62: Profinet Diagnostic ENC 2374P1
   RUNG wire#powerrail
      #PnDiag_ENC_2374P1(HW_IODevice := "2374P1~IODevice", Alarm := #Alarm.PnDiag_ENC_2374P1)
   END_RUNG
   // the same network as SCL:
   #PnDiag_ENC_2374P1(HW_IODevice := "2374P1~IODevice", Alarm := #Alarm.PnDiag_ENC_2374P1);   // "PnDiag"
END_REGION

REGION Network 63: Profinet Diagnostic ENC 2394P1
   RUNG wire#powerrail
      #PnDiag_ENC_2394P1(HW_IODevice := "2394P1~IODevice", Alarm := #Alarm.PnDiag_ENC_2394P1)
   END_RUNG
   // the same network as SCL:
   #PnDiag_ENC_2394P1(HW_IODevice := "2394P1~IODevice", Alarm := #Alarm.PnDiag_ENC_2394P1);   // "PnDiag"
END_REGION

REGION Network 64: Profinet Diagnostic ENC 2404P1
   RUNG wire#powerrail
      #PnDiag_ENC_2404P1(HW_IODevice := "2404P1~IODevice", Alarm := #Alarm.PnDiag_ENC_2404P1)
   END_RUNG
   // the same network as SCL:
   #PnDiag_ENC_2404P1(HW_IODevice := "2404P1~IODevice", Alarm := #Alarm.PnDiag_ENC_2404P1);   // "PnDiag"
END_REGION

REGION Network 65: Profinet Diagnostic ENC 2434P1
   RUNG wire#powerrail
      #PnDiag_ENC_2434P1(HW_IODevice := "2434P1~IODevice", Alarm := #Alarm.PnDiag_ENC_2434P1)
   END_RUNG
   // the same network as SCL:
   #PnDiag_ENC_2434P1(HW_IODevice := "2434P1~IODevice", Alarm := #Alarm.PnDiag_ENC_2434P1);   // "PnDiag"
END_REGION

REGION Network 66: Profinet Diagnostic ENC 2464P1
   RUNG wire#powerrail
      #PnDiag_ENC_2464P1(HW_IODevice := "2464P1~IODevice", Alarm := #Alarm.PnDiag_ENC_2464P1)
   END_RUNG
   // the same network as SCL:
   #PnDiag_ENC_2464P1(HW_IODevice := "2464P1~IODevice", Alarm := #Alarm.PnDiag_ENC_2464P1);   // "PnDiag"
END_REGION

REGION Network 67: Profinet Diagnostic ENC 2534P1
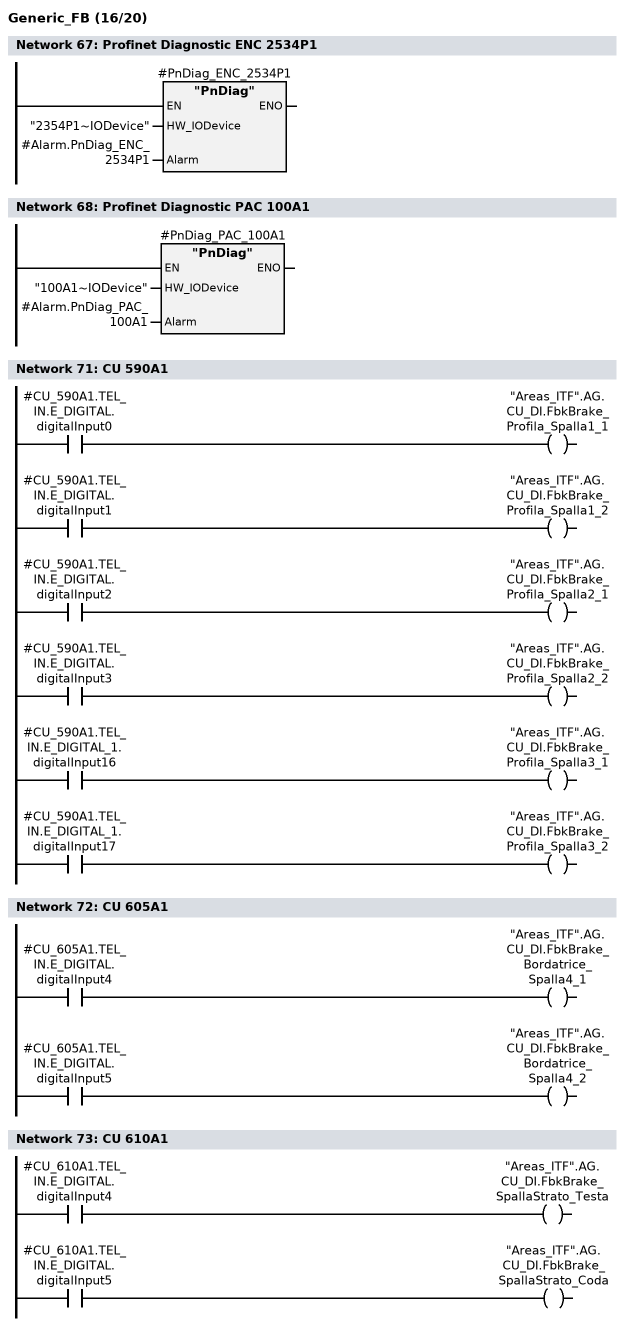
   RUNG wire#powerrail
      #PnDiag_ENC_2534P1(HW_IODevice := "2354P1~IODevice", Alarm := #Alarm.PnDiag_ENC_2534P1)
   END_RUNG
   // the same network as SCL:
   #PnDiag_ENC_2534P1(HW_IODevice := "2354P1~IODevice", Alarm := #Alarm.PnDiag_ENC_2534P1);   // "PnDiag"
END_REGION

REGION Network 68: Profinet Diagnostic PAC 100A1
   RUNG wire#powerrail
      #PnDiag_PAC_100A1(HW_IODevice := "100A1~IODevice", Alarm := #Alarm.PnDiag_PAC_100A1)
   END_RUNG
   // the same network as SCL:
   #PnDiag_PAC_100A1(HW_IODevice := "100A1~IODevice", Alarm := #Alarm.PnDiag_PAC_100A1);   // "PnDiag"
END_REGION

REGION Network 70: <<< CU DI >>>
END_REGION

REGION Network 71: CU 590A1
   RUNG wire#powerrail
      Contact( #CU_590A1.TEL_IN.E_DIGITAL.digitalInput0 )
      Coil( "Areas_ITF".AG.CU_DI.FbkBrake_Profila_Spalla1_1 )
   END_RUNG
   RUNG wire#powerrail
      Contact( #CU_590A1.TEL_IN.E_DIGITAL.digitalInput1 )
      Coil( "Areas_ITF".AG.CU_DI.FbkBrake_Profila_Spalla1_2 )
   END_RUNG
   RUNG wire#powerrail
      Contact( #CU_590A1.TEL_IN.E_DIGITAL.digitalInput2 )
      Coil( "Areas_ITF".AG.CU_DI.FbkBrake_Profila_Spalla2_1 )
   END_RUNG
   RUNG wire#powerrail
      Contact( #CU_590A1.TEL_IN.E_DIGITAL.digitalInput3 )
      Coil( "Areas_ITF".AG.CU_DI.FbkBrake_Profila_Spalla2_2 )
   END_RUNG
   RUNG wire#powerrail
      Contact( #CU_590A1.TEL_IN.E_DIGITAL_1.digitalInput16 )
      Coil( "Areas_ITF".AG.CU_DI.FbkBrake_Profila_Spalla3_1 )
   END_RUNG
   RUNG wire#powerrail
      Contact( #CU_590A1.TEL_IN.E_DIGITAL_1.digitalInput17 )
      Coil( "Areas_ITF".AG.CU_DI.FbkBrake_Profila_Spalla3_2 )
   END_RUNG
   // the same network as SCL:
   "Areas_ITF".AG.CU_DI.FbkBrake_Profila_Spalla1_1 := #CU_590A1.TEL_IN.E_DIGITAL.digitalInput0;
   "Areas_ITF".AG.CU_DI.FbkBrake_Profila_Spalla1_2 := #CU_590A1.TEL_IN.E_DIGITAL.digitalInput1;
   "Areas_ITF".AG.CU_DI.FbkBrake_Profila_Spalla2_1 := #CU_590A1.TEL_IN.E_DIGITAL.digitalInput2;
   "Areas_ITF".AG.CU_DI.FbkBrake_Profila_Spalla2_2 := #CU_590A1.TEL_IN.E_DIGITAL.digitalInput3;
   "Areas_ITF".AG.CU_DI.FbkBrake_Profila_Spalla3_1 := #CU_590A1.TEL_IN.E_DIGITAL_1.digitalInput16;
   "Areas_ITF".AG.CU_DI.FbkBrake_Profila_Spalla3_2 := #CU_590A1.TEL_IN.E_DIGITAL_1.digitalInput17;
END_REGION

REGION Network 72: CU 605A1
   RUNG wire#powerrail
      Contact( #CU_605A1.TEL_IN.E_DIGITAL.digitalInput4 )
      Coil( "Areas_ITF".AG.CU_DI.FbkBrake_Bordatrice_Spalla4_1 )
   END_RUNG
   RUNG wire#powerrail
      Contact( #CU_605A1.TEL_IN.E_DIGITAL.digitalInput5 )
      Coil( "Areas_ITF".AG.CU_DI.FbkBrake_Bordatrice_Spalla4_2 )
   END_RUNG
   // the same network as SCL:
   "Areas_ITF".AG.CU_DI.FbkBrake_Bordatrice_Spalla4_1 := #CU_605A1.TEL_IN.E_DIGITAL.digitalInput4;
   "Areas_ITF".AG.CU_DI.FbkBrake_Bordatrice_Spalla4_2 := #CU_605A1.TEL_IN.E_DIGITAL.digitalInput5;
END_REGION

REGION Network 73: CU 610A1
   RUNG wire#powerrail
      Contact( #CU_610A1.TEL_IN.E_DIGITAL.digitalInput4 )
      Coil( "Areas_ITF".AG.CU_DI.FbkBrake_SpallaStrato_Testa )
   END_RUNG
   RUNG wire#powerrail
      Contact( #CU_610A1.TEL_IN.E_DIGITAL.digitalInput5 )
      Coil( "Areas_ITF".AG.CU_DI.FbkBrake_SpallaStrato_Coda )
   END_RUNG
   // the same network as SCL:
   "Areas_ITF".AG.CU_DI.FbkBrake_SpallaStrato_Testa := #CU_610A1.TEL_IN.E_DIGITAL.digitalInput4;
   "Areas_ITF".AG.CU_DI.FbkBrake_SpallaStrato_Coda := #CU_610A1.TEL_IN.E_DIGITAL.digitalInput5;
END_REGION

REGION Network 74: CU 615A1
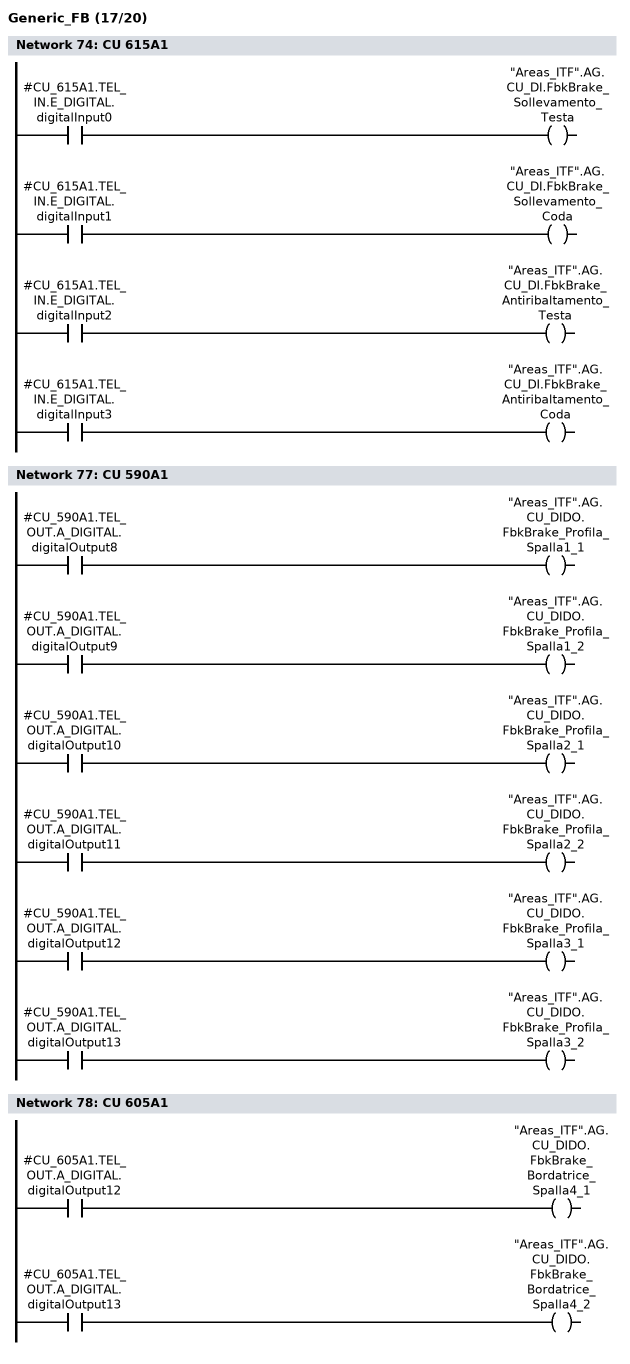
   RUNG wire#powerrail
      Contact( #CU_615A1.TEL_IN.E_DIGITAL.digitalInput0 )
      Coil( "Areas_ITF".AG.CU_DI.FbkBrake_Sollevamento_Testa )
   END_RUNG
   RUNG wire#powerrail
      Contact( #CU_615A1.TEL_IN.E_DIGITAL.digitalInput1 )
      Coil( "Areas_ITF".AG.CU_DI.FbkBrake_Sollevamento_Coda )
   END_RUNG
   RUNG wire#powerrail
      Contact( #CU_615A1.TEL_IN.E_DIGITAL.digitalInput2 )
      Coil( "Areas_ITF".AG.CU_DI.FbkBrake_Antiribaltamento_Testa )
   END_RUNG
   RUNG wire#powerrail
      Contact( #CU_615A1.TEL_IN.E_DIGITAL.digitalInput3 )
      Coil( "Areas_ITF".AG.CU_DI.FbkBrake_Antiribaltamento_Coda )
   END_RUNG
   // the same network as SCL:
   "Areas_ITF".AG.CU_DI.FbkBrake_Sollevamento_Testa := #CU_615A1.TEL_IN.E_DIGITAL.digitalInput0;
   "Areas_ITF".AG.CU_DI.FbkBrake_Sollevamento_Coda := #CU_615A1.TEL_IN.E_DIGITAL.digitalInput1;
   "Areas_ITF".AG.CU_DI.FbkBrake_Antiribaltamento_Testa := #CU_615A1.TEL_IN.E_DIGITAL.digitalInput2;
   "Areas_ITF".AG.CU_DI.FbkBrake_Antiribaltamento_Coda := #CU_615A1.TEL_IN.E_DIGITAL.digitalInput3;
END_REGION

REGION Network 76: <<< CU DI/DO >>>
END_REGION

REGION Network 77: CU 590A1
   RUNG wire#powerrail
      Contact( #CU_590A1.TEL_OUT.A_DIGITAL.digitalOutput8 )
      Coil( "Areas_ITF".AG.CU_DIDO.FbkBrake_Profila_Spalla1_1 )
   END_RUNG
   RUNG wire#powerrail
      Contact( #CU_590A1.TEL_OUT.A_DIGITAL.digitalOutput9 )
      Coil( "Areas_ITF".AG.CU_DIDO.FbkBrake_Profila_Spalla1_2 )
   END_RUNG
   RUNG wire#powerrail
      Contact( #CU_590A1.TEL_OUT.A_DIGITAL.digitalOutput10 )
      Coil( "Areas_ITF".AG.CU_DIDO.FbkBrake_Profila_Spalla2_1 )
   END_RUNG
   RUNG wire#powerrail
      Contact( #CU_590A1.TEL_OUT.A_DIGITAL.digitalOutput11 )
      Coil( "Areas_ITF".AG.CU_DIDO.FbkBrake_Profila_Spalla2_2 )
   END_RUNG
   RUNG wire#powerrail
      Contact( #CU_590A1.TEL_OUT.A_DIGITAL.digitalOutput12 )
      Coil( "Areas_ITF".AG.CU_DIDO.FbkBrake_Profila_Spalla3_1 )
   END_RUNG
   RUNG wire#powerrail
      Contact( #CU_590A1.TEL_OUT.A_DIGITAL.digitalOutput13 )
      Coil( "Areas_ITF".AG.CU_DIDO.FbkBrake_Profila_Spalla3_2 )
   END_RUNG
   // the same network as SCL:
   "Areas_ITF".AG.CU_DIDO.FbkBrake_Profila_Spalla1_1 := #CU_590A1.TEL_OUT.A_DIGITAL.digitalOutput8;
   "Areas_ITF".AG.CU_DIDO.FbkBrake_Profila_Spalla1_2 := #CU_590A1.TEL_OUT.A_DIGITAL.digitalOutput9;
   "Areas_ITF".AG.CU_DIDO.FbkBrake_Profila_Spalla2_1 := #CU_590A1.TEL_OUT.A_DIGITAL.digitalOutput10;
   "Areas_ITF".AG.CU_DIDO.FbkBrake_Profila_Spalla2_2 := #CU_590A1.TEL_OUT.A_DIGITAL.digitalOutput11;
   "Areas_ITF".AG.CU_DIDO.FbkBrake_Profila_Spalla3_1 := #CU_590A1.TEL_OUT.A_DIGITAL.digitalOutput12;
   "Areas_ITF".AG.CU_DIDO.FbkBrake_Profila_Spalla3_2 := #CU_590A1.TEL_OUT.A_DIGITAL.digitalOutput13;
END_REGION

REGION Network 78: CU 605A1
   RUNG wire#powerrail
      Contact( #CU_605A1.TEL_OUT.A_DIGITAL.digitalOutput12 )
      Coil( "Areas_ITF".AG.CU_DIDO.FbkBrake_Bordatrice_Spalla4_1 )
   END_RUNG
   RUNG wire#powerrail
      Contact( #CU_605A1.TEL_OUT.A_DIGITAL.digitalOutput13 )
      Coil( "Areas_ITF".AG.CU_DIDO.FbkBrake_Bordatrice_Spalla4_2 )
   END_RUNG
   // the same network as SCL:
   "Areas_ITF".AG.CU_DIDO.FbkBrake_Bordatrice_Spalla4_1 := #CU_605A1.TEL_OUT.A_DIGITAL.digitalOutput12;
   "Areas_ITF".AG.CU_DIDO.FbkBrake_Bordatrice_Spalla4_2 := #CU_605A1.TEL_OUT.A_DIGITAL.digitalOutput13;
END_REGION

REGION Network 79: CU 610A1
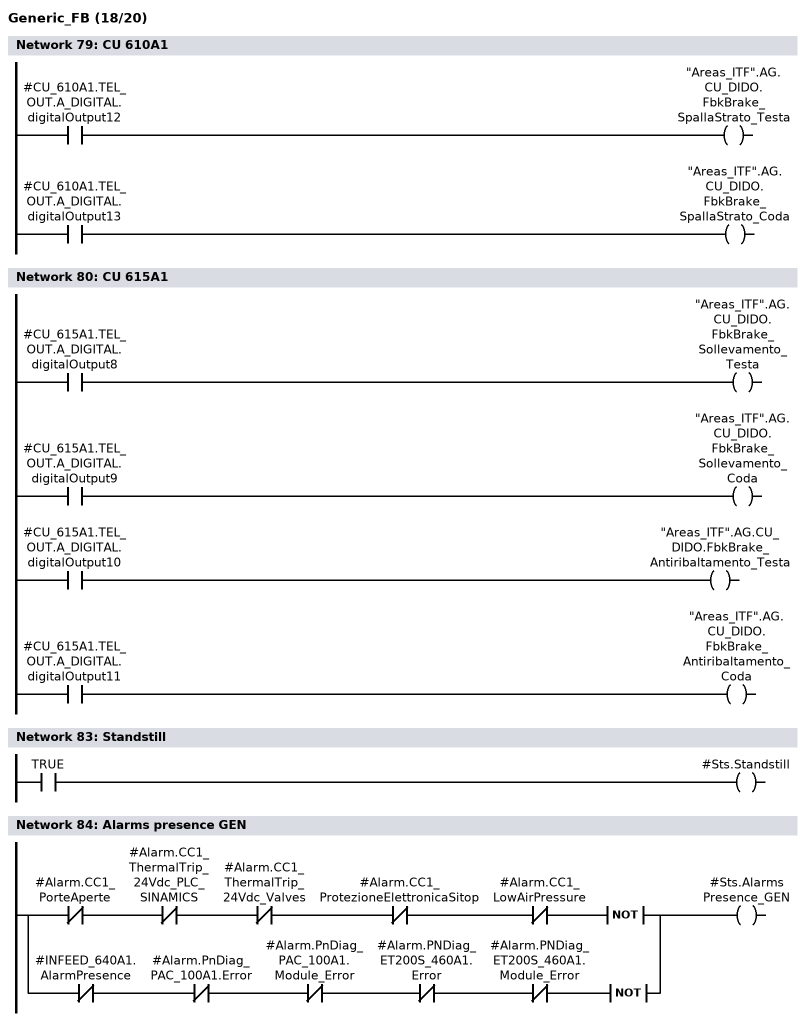
   RUNG wire#powerrail
      Contact( #CU_610A1.TEL_OUT.A_DIGITAL.digitalOutput12 )
      Coil( "Areas_ITF".AG.CU_DIDO.FbkBrake_SpallaStrato_Testa )
   END_RUNG
   RUNG wire#powerrail
      Contact( #CU_610A1.TEL_OUT.A_DIGITAL.digitalOutput13 )
      Coil( "Areas_ITF".AG.CU_DIDO.FbkBrake_SpallaStrato_Coda )
   END_RUNG
   // the same network as SCL:
   "Areas_ITF".AG.CU_DIDO.FbkBrake_SpallaStrato_Testa := #CU_610A1.TEL_OUT.A_DIGITAL.digitalOutput12;
   "Areas_ITF".AG.CU_DIDO.FbkBrake_SpallaStrato_Coda := #CU_610A1.TEL_OUT.A_DIGITAL.digitalOutput13;
END_REGION

REGION Network 80: CU 615A1
   RUNG wire#powerrail
      Contact( #CU_615A1.TEL_OUT.A_DIGITAL.digitalOutput8 )
      Coil( "Areas_ITF".AG.CU_DIDO.FbkBrake_Sollevamento_Testa )
   END_RUNG
   RUNG wire#powerrail
      Contact( #CU_615A1.TEL_OUT.A_DIGITAL.digitalOutput9 )
      Coil( "Areas_ITF".AG.CU_DIDO.FbkBrake_Sollevamento_Coda )
   END_RUNG
   RUNG wire#powerrail
      Contact( #CU_615A1.TEL_OUT.A_DIGITAL.digitalOutput10 )
      Coil( "Areas_ITF".AG.CU_DIDO.FbkBrake_Antiribaltamento_Testa )
   END_RUNG
   RUNG wire#powerrail
      Contact( #CU_615A1.TEL_OUT.A_DIGITAL.digitalOutput11 )
      Coil( "Areas_ITF".AG.CU_DIDO.FbkBrake_Antiribaltamento_Coda )
   END_RUNG
   // the same network as SCL:
   "Areas_ITF".AG.CU_DIDO.FbkBrake_Sollevamento_Testa := #CU_615A1.TEL_OUT.A_DIGITAL.digitalOutput8;
   "Areas_ITF".AG.CU_DIDO.FbkBrake_Sollevamento_Coda := #CU_615A1.TEL_OUT.A_DIGITAL.digitalOutput9;
   "Areas_ITF".AG.CU_DIDO.FbkBrake_Antiribaltamento_Testa := #CU_615A1.TEL_OUT.A_DIGITAL.digitalOutput10;
   "Areas_ITF".AG.CU_DIDO.FbkBrake_Antiribaltamento_Coda := #CU_615A1.TEL_OUT.A_DIGITAL.digitalOutput11;
END_REGION

REGION Network 82: <<< MACHINE STATUS >>>
END_REGION

REGION Network 83: Standstill
   RUNG wire#powerrail
      Contact( TRUE )
      Coil( #Sts.Standstill )
   END_RUNG
   // the same network as SCL:
   #Sts.Standstill := TRUE;
END_REGION

REGION Network 84: Alarms presence GEN
   RUNG wire#powerrail
      I_Contact( #Alarm.CC1_PorteAperte )
      I_Contact( #Alarm.CC1_ThermalTrip_24Vdc_PLC_SINAMICS )
      I_Contact( #Alarm.CC1_ThermalTrip_24Vdc_Valves )
      I_Contact( #Alarm.CC1_ProtezioneElettronicaSitop )
      I_Contact( #Alarm.CC1_LowAirPressure )
      Not()
      wire#w1
      Coil( #Sts.AlarmsPresence_GEN )
   END_RUNG
   RUNG wire#powerrail
      I_Contact( #INFEED_640A1.AlarmPresence )
      I_Contact( #Alarm.PnDiag_PAC_100A1.Error )
      I_Contact( #Alarm.PnDiag_PAC_100A1.Module_Error )
      I_Contact( #Alarm.PNDiag_ET200S_460A1.Error )
      I_Contact( #Alarm.PNDiag_ET200S_460A1.Module_Error )
      Not()
   END_RUNG wire#w1
   // the same network as SCL:
   #Sts.AlarmsPresence_GEN := NOT (NOT #Alarm.CC1_PorteAperte AND NOT #Alarm.CC1_ThermalTrip_24Vdc_PLC_SINAMICS AND NOT #Alarm.CC1_ThermalTrip_24Vdc_Valves AND NOT #Alarm.CC1_ProtezioneElettronicaSitop AND NOT #Alarm.CC1_LowAirPressure) OR NOT (NOT #INFEED_640A1.AlarmPresence AND NOT #Alarm.PnDiag_PAC_100A1.Error AND NOT #Alarm.PnDiag_PAC_100A1.Module_Error AND NOT #Alarm.PNDiag_ET200S_460A1.Error AND NOT #Alarm.PNDiag_ET200S_460A1.Module_Error);
END_REGION

REGION Network 85: Alarms presence A01 A02
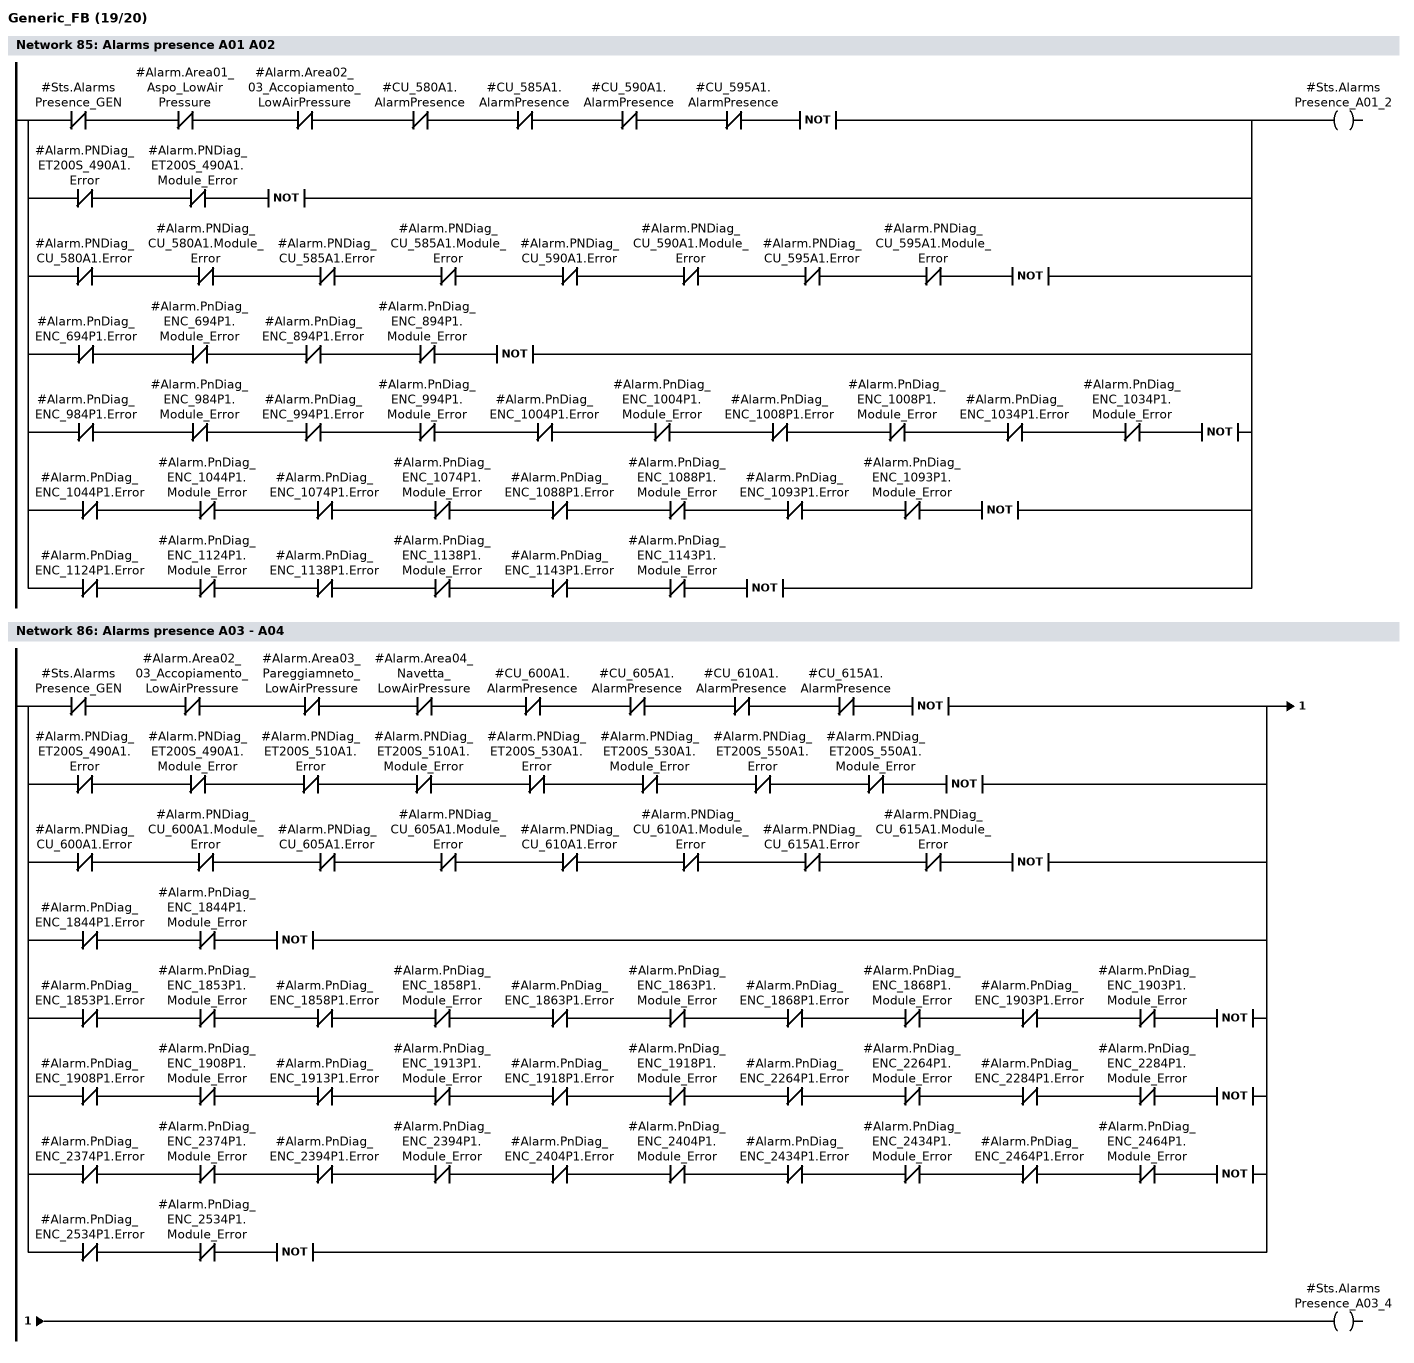
   RUNG wire#powerrail
      I_Contact( #Sts.AlarmsPresence_GEN )
      I_Contact( #Alarm.Area01_Aspo_LowAirPressure )
      I_Contact( #Alarm.Area02_03_Accopiamento_LowAirPressure )
      I_Contact( #CU_580A1.AlarmPresence )
      I_Contact( #CU_585A1.AlarmPresence )
      I_Contact( #CU_590A1.AlarmPresence )
      I_Contact( #CU_595A1.AlarmPresence )
      Not()
      wire#w1
      Coil( #Sts.AlarmsPresence_A01_2 )
   END_RUNG
   RUNG wire#powerrail
      I_Contact( #Alarm.PNDiag_ET200S_490A1.Error )
      I_Contact( #Alarm.PNDiag_ET200S_490A1.Module_Error )
      Not()
   END_RUNG wire#w1
   RUNG wire#powerrail
      I_Contact( #Alarm.PNDiag_CU_580A1.Error )
      I_Contact( #Alarm.PNDiag_CU_580A1.Module_Error )
      I_Contact( #Alarm.PNDiag_CU_585A1.Error )
      I_Contact( #Alarm.PNDiag_CU_585A1.Module_Error )
      I_Contact( #Alarm.PNDiag_CU_590A1.Error )
      I_Contact( #Alarm.PNDiag_CU_590A1.Module_Error )
      I_Contact( #Alarm.PNDiag_CU_595A1.Error )
      I_Contact( #Alarm.PNDiag_CU_595A1.Module_Error )
      Not()
   END_RUNG wire#w1
   RUNG wire#powerrail
      I_Contact( #Alarm.PnDiag_ENC_694P1.Error )
      I_Contact( #Alarm.PnDiag_ENC_694P1.Module_Error )
      I_Contact( #Alarm.PnDiag_ENC_894P1.Error )
      I_Contact( #Alarm.PnDiag_ENC_894P1.Module_Error )
      Not()
   END_RUNG wire#w1
   RUNG wire#powerrail
      I_Contact( #Alarm.PnDiag_ENC_984P1.Error )
      I_Contact( #Alarm.PnDiag_ENC_984P1.Module_Error )
      I_Contact( #Alarm.PnDiag_ENC_994P1.Error )
      I_Contact( #Alarm.PnDiag_ENC_994P1.Module_Error )
      I_Contact( #Alarm.PnDiag_ENC_1004P1.Error )
      I_Contact( #Alarm.PnDiag_ENC_1004P1.Module_Error )
      I_Contact( #Alarm.PnDiag_ENC_1008P1.Error )
      I_Contact( #Alarm.PnDiag_ENC_1008P1.Module_Error )
      I_Contact( #Alarm.PnDiag_ENC_1034P1.Error )
      I_Contact( #Alarm.PnDiag_ENC_1034P1.Module_Error )
      Not()
   END_RUNG wire#w1
   RUNG wire#powerrail
      I_Contact( #Alarm.PnDiag_ENC_1044P1.Error )
      I_Contact( #Alarm.PnDiag_ENC_1044P1.Module_Error )
      I_Contact( #Alarm.PnDiag_ENC_1074P1.Error )
      I_Contact( #Alarm.PnDiag_ENC_1074P1.Module_Error )
      I_Contact( #Alarm.PnDiag_ENC_1088P1.Error )
      I_Contact( #Alarm.PnDiag_ENC_1088P1.Module_Error )
      I_Contact( #Alarm.PnDiag_ENC_1093P1.Error )
      I_Contact( #Alarm.PnDiag_ENC_1093P1.Module_Error )
      Not()
   END_RUNG wire#w1
   RUNG wire#powerrail
      I_Contact( #Alarm.PnDiag_ENC_1124P1.Error )
      I_Contact( #Alarm.PnDiag_ENC_1124P1.Module_Error )
      I_Contact( #Alarm.PnDiag_ENC_1138P1.Error )
      I_Contact( #Alarm.PnDiag_ENC_1138P1.Module_Error )
      I_Contact( #Alarm.PnDiag_ENC_1143P1.Error )
      I_Contact( #Alarm.PnDiag_ENC_1143P1.Module_Error )
      Not()
   END_RUNG wire#w1
   // the same network as SCL:
   #Sts.AlarmsPresence_A01_2 := NOT (NOT #Sts.AlarmsPresence_GEN AND NOT #Alarm.Area01_Aspo_LowAirPressure AND NOT #Alarm.Area02_03_Accopiamento_LowAirPressure AND NOT #CU_580A1.AlarmPresence AND NOT #CU_585A1.AlarmPresence AND NOT #CU_590A1.AlarmPresence AND NOT #CU_595A1.AlarmPresence) OR NOT (NOT #Alarm.PNDiag_ET200S_490A1.Error AND NOT #Alarm.PNDiag_ET200S_490A1.Module_Error) OR NOT (NOT #Alarm.PNDiag_CU_580A1.Error AND NOT #Alarm.PNDiag_CU_580A1.Module_Error AND NOT #Alarm.PNDiag_CU_585A1.Error AND NOT #Alarm.PNDiag_CU_585A1.Module_Error AND NOT #Alarm.PNDiag_CU_590A1.Error AND NOT #Alarm.PNDiag_CU_590A1.Module_Error AND NOT #Alarm.PNDiag_CU_595A1.Error AND NOT #Alarm.PNDiag_CU_595A1.Module_Error) OR NOT (NOT #Alarm.PnDiag_ENC_694P1.Error AND NOT #Alarm.PnDiag_ENC_694P1.Module_Error AND NOT #Alarm.PnDiag_ENC_894P1.Error AND NOT #Alarm.PnDiag_ENC_894P1.Module_Error) OR NOT (NOT #Alarm.PnDiag_ENC_984P1.Error AND NOT #Alarm.PnDiag_ENC_984P1.Module_Error AND NOT #Alarm.PnDiag_ENC_994P1.Error AND NOT #Alarm.PnDiag_ENC_994P1.Module_Error AND NOT #Alarm.PnDiag_ENC_1004P1.Error AND NOT #Alarm.PnDiag_ENC_1004P1.Module_Error AND NOT #Alarm.PnDiag_ENC_1008P1.Error AND NOT #Alarm.PnDiag_ENC_1008P1.Module_Error AND NOT #Alarm.PnDiag_ENC_1034P1.Error AND NOT #Alarm.PnDiag_ENC_1034P1.Module_Error) OR NOT (NOT #Alarm.PnDiag_ENC_1044P1.Error AND NOT #Alarm.PnDiag_ENC_1044P1.Module_Error AND NOT #Alarm.PnDiag_ENC_1074P1.Error AND NOT #Alarm.PnDiag_ENC_1074P1.Module_Error AND NOT #Alarm.PnDiag_ENC_1088P1.Error AND NOT #Alarm.PnDiag_ENC_1088P1.Module_Error AND NOT #Alarm.PnDiag_ENC_1093P1.Error AND NOT #Alarm.PnDiag_ENC_1093P1.Module_Error) OR NOT (NOT #Alarm.PnDiag_ENC_1124P1.Error AND NOT #Alarm.PnDiag_ENC_1124P1.Module_Error AND NOT #Alarm.PnDiag_ENC_1138P1.Error AND NOT #Alarm.PnDiag_ENC_1138P1.Module_Error AND NOT #Alarm.PnDiag_ENC_1143P1.Error AND NOT #Alarm.PnDiag_ENC_1143P1.Module_Error);
END_REGION

REGION Network 86: Alarms presence A03 - A04
   RUNG wire#powerrail
      I_Contact( #Sts.AlarmsPresence_GEN )
      I_Contact( #Alarm.Area02_03_Accopiamento_LowAirPressure )
      I_Contact( #Alarm.Area03_Pareggiamneto_LowAirPressure )
      I_Contact( #Alarm.Area04_Navetta_LowAirPressure )
      I_Contact( #CU_600A1.AlarmPresence )
      I_Contact( #CU_605A1.AlarmPresence )
      I_Contact( #CU_610A1.AlarmPresence )
      I_Contact( #CU_615A1.AlarmPresence )
      Not()
      wire#w1
      Coil( #Sts.AlarmsPresence_A03_4 )
   END_RUNG
   RUNG wire#powerrail
      I_Contact( #Alarm.PNDiag_ET200S_490A1.Error )
      I_Contact( #Alarm.PNDiag_ET200S_490A1.Module_Error )
      I_Contact( #Alarm.PNDiag_ET200S_510A1.Error )
      I_Contact( #Alarm.PNDiag_ET200S_510A1.Module_Error )
      I_Contact( #Alarm.PNDiag_ET200S_530A1.Error )
      I_Contact( #Alarm.PNDiag_ET200S_530A1.Module_Error )
      I_Contact( #Alarm.PNDiag_ET200S_550A1.Error )
      I_Contact( #Alarm.PNDiag_ET200S_550A1.Module_Error )
      Not()
   END_RUNG wire#w1
   RUNG wire#powerrail
      I_Contact( #Alarm.PNDiag_CU_600A1.Error )
      I_Contact( #Alarm.PNDiag_CU_600A1.Module_Error )
      I_Contact( #Alarm.PNDiag_CU_605A1.Error )
      I_Contact( #Alarm.PNDiag_CU_605A1.Module_Error )
      I_Contact( #Alarm.PNDiag_CU_610A1.Error )
      I_Contact( #Alarm.PNDiag_CU_610A1.Module_Error )
      I_Contact( #Alarm.PNDiag_CU_615A1.Error )
      I_Contact( #Alarm.PNDiag_CU_615A1.Module_Error )
      Not()
   END_RUNG wire#w1
   RUNG wire#powerrail
      I_Contact( #Alarm.PnDiag_ENC_1844P1.Error )
      I_Contact( #Alarm.PnDiag_ENC_1844P1.Module_Error )
      Not()
   END_RUNG wire#w1
   RUNG wire#powerrail
      I_Contact( #Alarm.PnDiag_ENC_1853P1.Error )
      I_Contact( #Alarm.PnDiag_ENC_1853P1.Module_Error )
      I_Contact( #Alarm.PnDiag_ENC_1858P1.Error )
      I_Contact( #Alarm.PnDiag_ENC_1858P1.Module_Error )
      I_Contact( #Alarm.PnDiag_ENC_1863P1.Error )
      I_Contact( #Alarm.PnDiag_ENC_1863P1.Module_Error )
      I_Contact( #Alarm.PnDiag_ENC_1868P1.Error )
      I_Contact( #Alarm.PnDiag_ENC_1868P1.Module_Error )
      I_Contact( #Alarm.PnDiag_ENC_1903P1.Error )
      I_Contact( #Alarm.PnDiag_ENC_1903P1.Module_Error )
      Not()
   END_RUNG wire#w1
   RUNG wire#powerrail
      I_Contact( #Alarm.PnDiag_ENC_1908P1.Error )
      I_Contact( #Alarm.PnDiag_ENC_1908P1.Module_Error )
      I_Contact( #Alarm.PnDiag_ENC_1913P1.Error )
      I_Contact( #Alarm.PnDiag_ENC_1913P1.Module_Error )
      I_Contact( #Alarm.PnDiag_ENC_1918P1.Error )
      I_Contact( #Alarm.PnDiag_ENC_1918P1.Module_Error )
      I_Contact( #Alarm.PnDiag_ENC_2264P1.Error )
      I_Contact( #Alarm.PnDiag_ENC_2264P1.Module_Error )
      I_Contact( #Alarm.PnDiag_ENC_2284P1.Error )
      I_Contact( #Alarm.PnDiag_ENC_2284P1.Module_Error )
      Not()
   END_RUNG wire#w1
   RUNG wire#powerrail
      I_Contact( #Alarm.PnDiag_ENC_2374P1.Error )
      I_Contact( #Alarm.PnDiag_ENC_2374P1.Module_Error )
      I_Contact( #Alarm.PnDiag_ENC_2394P1.Error )
      I_Contact( #Alarm.PnDiag_ENC_2394P1.Module_Error )
      I_Contact( #Alarm.PnDiag_ENC_2404P1.Error )
      I_Contact( #Alarm.PnDiag_ENC_2404P1.Module_Error )
      I_Contact( #Alarm.PnDiag_ENC_2434P1.Error )
      I_Contact( #Alarm.PnDiag_ENC_2434P1.Module_Error )
      I_Contact( #Alarm.PnDiag_ENC_2464P1.Error )
      I_Contact( #Alarm.PnDiag_ENC_2464P1.Module_Error )
      Not()
   END_RUNG wire#w1
   RUNG wire#powerrail
      I_Contact( #Alarm.PnDiag_ENC_2534P1.Error )
      I_Contact( #Alarm.PnDiag_ENC_2534P1.Module_Error )
      Not()
   END_RUNG wire#w1
   // the same network as SCL:
   #Sts.AlarmsPresence_A03_4 := NOT (NOT #Sts.AlarmsPresence_GEN AND NOT #Alarm.Area02_03_Accopiamento_LowAirPressure AND NOT #Alarm.Area03_Pareggiamneto_LowAirPressure AND NOT #Alarm.Area04_Navetta_LowAirPressure AND NOT #CU_600A1.AlarmPresence AND NOT #CU_605A1.AlarmPresence AND NOT #CU_610A1.AlarmPresence AND NOT #CU_615A1.AlarmPresence) OR NOT (NOT #Alarm.PNDiag_ET200S_490A1.Error AND NOT #Alarm.PNDiag_ET200S_490A1.Module_Error AND NOT #Alarm.PNDiag_ET200S_510A1.Error AND NOT #Alarm.PNDiag_ET200S_510A1.Module_Error AND NOT #Alarm.PNDiag_ET200S_530A1.Error AND NOT #Alarm.PNDiag_ET200S_530A1.Module_Error AND NOT #Alarm.PNDiag_ET200S_550A1.Error AND NOT #Alarm.PNDiag_ET200S_550A1.Module_Error) OR NOT (NOT #Alarm.PNDiag_CU_600A1.Error AND NOT #Alarm.PNDiag_CU_600A1.Module_Error AND NOT #Alarm.PNDiag_CU_605A1.Error AND NOT #Alarm.PNDiag_CU_605A1.Module_Error AND NOT #Alarm.PNDiag_CU_610A1.Error AND NOT #Alarm.PNDiag_CU_610A1.Module_Error AND NOT #Alarm.PNDiag_CU_615A1.Error AND NOT #Alarm.PNDiag_CU_615A1.Module_Error) OR NOT (NOT #Alarm.PnDiag_ENC_1844P1.Error AND NOT #Alarm.PnDiag_ENC_1844P1.Module_Error) OR NOT (NOT #Alarm.PnDiag_ENC_1853P1.Error AND NOT #Alarm.PnDiag_ENC_1853P1.Module_Error AND NOT #Alarm.PnDiag_ENC_1858P1.Error AND NOT #Alarm.PnDiag_ENC_1858P1.Module_Error AND NOT #Alarm.PnDiag_ENC_1863P1.Error AND NOT #Alarm.PnDiag_ENC_1863P1.Module_Error AND NOT #Alarm.PnDiag_ENC_1868P1.Error AND NOT #Alarm.PnDiag_ENC_1868P1.Module_Error AND NOT #Alarm.PnDiag_ENC_1903P1.Error AND NOT #Alarm.PnDiag_ENC_1903P1.Module_Error) OR NOT (NOT #Alarm.PnDiag_ENC_1908P1.Error AND NOT #Alarm.PnDiag_ENC_1908P1.Module_Error AND NOT #Alarm.PnDiag_ENC_1913P1.Error AND NOT #Alarm.PnDiag_ENC_1913P1.Module_Error AND NOT #Alarm.PnDiag_ENC_1918P1.Error AND NOT #Alarm.PnDiag_ENC_1918P1.Module_Error AND NOT #Alarm.PnDiag_ENC_2264P1.Error AND NOT #Alarm.PnDiag_ENC_2264P1.Module_Error AND NOT #Alarm.PnDiag_ENC_2284P1.Error AND NOT #Alarm.PnDiag_ENC_2284P1.Module_Error) OR NOT (NOT #Alarm.PnDiag_ENC_2374P1.Error AND NOT #Alarm.PnDiag_ENC_2374P1.Module_Error AND NOT #Alarm.PnDiag_ENC_2394P1.Error AND NOT #Alarm.PnDiag_ENC_2394P1.Module_Error AND NOT #Alarm.PnDiag_ENC_2404P1.Error AND NOT #Alarm.PnDiag_ENC_2404P1.Module_Error AND NOT #Alarm.PnDiag_ENC_2434P1.Error AND NOT #Alarm.PnDiag_ENC_2434P1.Module_Error AND NOT #Alarm.PnDiag_ENC_2464P1.Error AND NOT #Alarm.PnDiag_ENC_2464P1.Module_Error) OR NOT (NOT #Alarm.PnDiag_ENC_2534P1.Error AND NOT #Alarm.PnDiag_ENC_2534P1.Module_Error);
END_REGION

REGION Network 87: Warnings presence
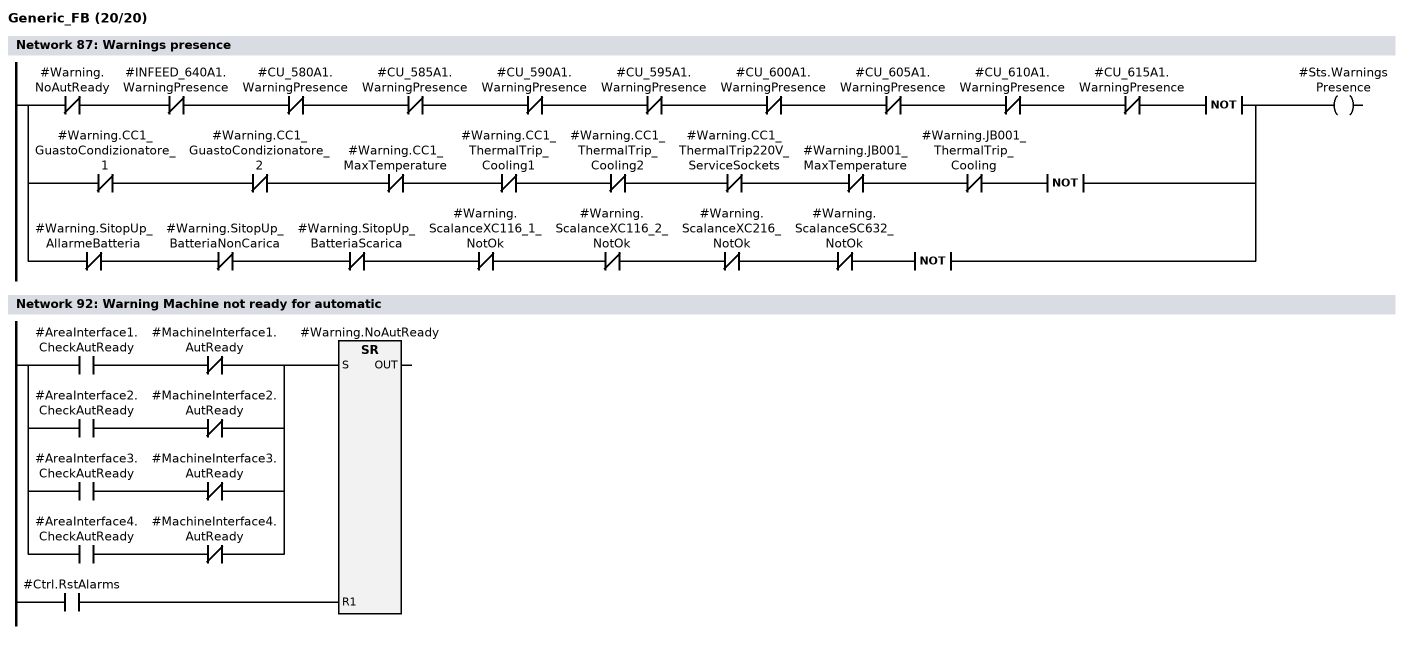
   RUNG wire#powerrail
      I_Contact( #Warning.NoAutReady )
      I_Contact( #INFEED_640A1.WarningPresence )
      I_Contact( #CU_580A1.WarningPresence )
      I_Contact( #CU_585A1.WarningPresence )
      I_Contact( #CU_590A1.WarningPresence )
      I_Contact( #CU_595A1.WarningPresence )
      I_Contact( #CU_600A1.WarningPresence )
      I_Contact( #CU_605A1.WarningPresence )
      I_Contact( #CU_610A1.WarningPresence )
      I_Contact( #CU_615A1.WarningPresence )
      Not()
      wire#w1
      Coil( #Sts.WarningsPresence )
   END_RUNG
   RUNG wire#powerrail
      I_Contact( #Warning.CC1_GuastoCondizionatore_1 )
      I_Contact( #Warning.CC1_GuastoCondizionatore_2 )
      I_Contact( #Warning.CC1_MaxTemperature )
      I_Contact( #Warning.CC1_ThermalTrip_Cooling1 )
      I_Contact( #Warning.CC1_ThermalTrip_Cooling2 )
      I_Contact( #Warning.CC1_ThermalTrip220V_ServiceSockets )
      I_Contact( #Warning.JB001_MaxTemperature )
      I_Contact( #Warning.JB001_ThermalTrip_Cooling )
      Not()
   END_RUNG wire#w1
   RUNG wire#powerrail
      I_Contact( #Warning.SitopUp_AllarmeBatteria )
      I_Contact( #Warning.SitopUp_BatteriaNonCarica )
      I_Contact( #Warning.SitopUp_BatteriaScarica )
      I_Contact( #Warning.ScalanceXC116_1_NotOk )
      I_Contact( #Warning.ScalanceXC116_2_NotOk )
      I_Contact( #Warning.ScalanceXC216_NotOk )
      I_Contact( #Warning.ScalanceSC632_NotOk )
      Not()
   END_RUNG wire#w1
   // the same network as SCL:
   #Sts.WarningsPresence := NOT (NOT #Warning.NoAutReady AND NOT #INFEED_640A1.WarningPresence AND NOT #CU_580A1.WarningPresence AND NOT #CU_585A1.WarningPresence AND NOT #CU_590A1.WarningPresence AND NOT #CU_595A1.WarningPresence AND NOT #CU_600A1.WarningPresence AND NOT #CU_605A1.WarningPresence AND NOT #CU_610A1.WarningPresence AND NOT #CU_615A1.WarningPresence) OR NOT (NOT #Warning.CC1_GuastoCondizionatore_1 AND NOT #Warning.CC1_GuastoCondizionatore_2 AND NOT #Warning.CC1_MaxTemperature AND NOT #Warning.CC1_ThermalTrip_Cooling1 AND NOT #Warning.CC1_ThermalTrip_Cooling2 AND NOT #Warning.CC1_ThermalTrip220V_ServiceSockets AND NOT #Warning.JB001_MaxTemperature AND NOT #Warning.JB001_ThermalTrip_Cooling) OR NOT (NOT #Warning.SitopUp_AllarmeBatteria AND NOT #Warning.SitopUp_BatteriaNonCarica AND NOT #Warning.SitopUp_BatteriaScarica AND NOT #Warning.ScalanceXC116_1_NotOk AND NOT #Warning.ScalanceXC116_2_NotOk AND NOT #Warning.ScalanceXC216_NotOk AND NOT #Warning.ScalanceSC632_NotOk);
END_REGION

REGION Network 88 (SCL): Collect machine to zone interface 1
   #MachineInterface1.AutReady := #AreaInterface1.Aut AND NOT #Sts.AlarmsPresence_A01_2;
   #MachineInterface1.Aborting := #Sts.AlarmsPresence_A01_2;
   #MachineInterface1.MotionsStandStill := #Sts.Standstill;
   #MachineInterface1.AckStopInPhase := #AreaInterface1.StopInPhase;
   #MachineInterface1.AckStopProgrammed := #AreaInterface1.StopProgrammed;
   #MachineInterface1.AlarmsPresence := #Sts.AlarmsPresence_A01_2;
   #MachineInterface1.WarningPresence := #Sts.WarningsPresence;
END_REGION

REGION Network 89 (SCL): Collect machine to zone interface 2
   #MachineInterface2.AutReady := #AreaInterface2.Aut AND NOT #Sts.AlarmsPresence_A01_2;
   #MachineInterface2.Aborting := #Sts.AlarmsPresence_A01_2;
   #MachineInterface2.MotionsStandStill := #Sts.Standstill;
   #MachineInterface2.AckStopInPhase := #AreaInterface2.StopInPhase;
   #MachineInterface2.AckStopProgrammed := #AreaInterface2.StopProgrammed;
   #MachineInterface2.AlarmsPresence := #Sts.AlarmsPresence_A01_2;
   #MachineInterface2.WarningPresence := #Sts.WarningsPresence;
END_REGION

REGION Network 90 (SCL): Collect machine to zone interface 3
   #MachineInterface3.AutReady := #AreaInterface3.Aut AND NOT #Sts.AlarmsPresence_A03_4;
   #MachineInterface3.Aborting := #Sts.AlarmsPresence_A03_4;
   #MachineInterface3.MotionsStandStill := #Sts.Standstill;
   #MachineInterface3.AckStopInPhase := #AreaInterface3.StopInPhase;
   #MachineInterface3.AckStopProgrammed := #AreaInterface3.StopProgrammed;
   #MachineInterface3.AlarmsPresence := #Sts.AlarmsPresence_A03_4;
   #MachineInterface3.WarningPresence := #Sts.WarningsPresence;
END_REGION

REGION Network 91 (SCL): Collect machine to zone interface 4
   #MachineInterface3.AutReady := #AreaInterface4.Aut AND NOT #Sts.AlarmsPresence_A03_4;
   #MachineInterface3.Aborting := #Sts.AlarmsPresence_A03_4;
   #MachineInterface3.MotionsStandStill := #Sts.Standstill;
   #MachineInterface3.AckStopInPhase := #AreaInterface4.StopInPhase;
   #MachineInterface3.AckStopProgrammed := #AreaInterface4.StopProgrammed;
   #MachineInterface3.AlarmsPresence := #Sts.AlarmsPresence_A03_4;
   #MachineInterface3.WarningPresence := #Sts.WarningsPresence;
END_REGION

REGION Network 92: Warning Machine not ready for automatic
   RUNG wire#powerrail
      Contact( #AreaInterface1.CheckAutReady )
      I_Contact( #MachineInterface1.AutReady )
      wire#w1
      S_SR(operand := #Warning.NoAutReady, r1 := wire#w2)
   END_RUNG
   RUNG wire#powerrail
      Contact( #AreaInterface2.CheckAutReady )
      I_Contact( #MachineInterface2.AutReady )
   END_RUNG wire#w1
   RUNG wire#powerrail
      Contact( #AreaInterface3.CheckAutReady )
      I_Contact( #MachineInterface3.AutReady )
   END_RUNG wire#w1
   RUNG wire#powerrail
      Contact( #AreaInterface4.CheckAutReady )
      I_Contact( #MachineInterface4.AutReady )
   END_RUNG wire#w1
   RUNG wire#powerrail
      Contact( #Ctrl.RstAlarms )
   END_RUNG wire#w2
   // the same network as SCL:
   IF (#AreaInterface1.CheckAutReady AND NOT #MachineInterface1.AutReady) OR (#AreaInterface2.CheckAutReady AND NOT #MachineInterface2.AutReady) OR (#AreaInterface3.CheckAutReady AND NOT #MachineInterface3.AutReady) OR (#AreaInterface4.CheckAutReady AND NOT #MachineInterface4.AutReady) THEN
       #Warning.NoAutReady := TRUE;   // SR flip-flop
   END_IF;
   IF #Ctrl.RstAlarms THEN #Warning.NoAutReady := FALSE; END_IF;
END_REGION

REGION Network 93: >
END_REGION

REGION Network 94: >
END_REGION
END_FUNCTION_BLOCK
